# B&R Automation Studio project EFI (part 20)

#### MachineCtrl_Slow.var
```iecst
VAR
	iPrimerBarMechanicalPosition : USINT; (*Position of white bar regarding mechanical assembly*)
	iPrimerBarMapping : USINT; (*Position of white bar regarding printing definition in UI*)
	iWhiteBarMechanicalPosition : USINT; (*Position of white bar regarding mechanical assembly*)
	iWhiteBarMapping : USINT; (*Position of white bar regarding printing definition in UI*)
	arNotLoadedImage : AutoResetSound;
	arSAIFault : AutoResetSound;
	arBentTile : AutoResetSound;
	arPDSensorErrorL1 : AutoResetSound;
	arPDSensorErrorL2 : AutoResetSound;
	xAllBlocksCleaning : BOOL;
	xInstantPrintL2 : BOOL;
	xAllBlocksCleaningEnded : BOOL;
	xInstantPrintL1 : BOOL; (*command bool edge*)
	xShotLine2 : BOOL;
	xCleanSequencially : BOOL := FALSE;
	xShotLine1 : BOOL;
	xOrderToGap : BOOL;
	xCleanBeltForced : BOOL;
	xCleaningBeltByTiles : BOOL;
	xOutputConsentInSingleLineL1 : BOOL;
	xOutputConsentInByPassL1 : BOOL;
	xOutputConsentInByPassL2 : BOOL;
	xOutputConsentInDTPL1 : BOOL;
	xOutputConsentInDTPL2 : BOOL;
	xDoubleLineConsent : BOOL; (*Belt Consent in DobleLine Mode*)
	xOnPcs : BOOL;
	xCleaningBeltByTime : BOOL;
	xCleanBeltOrder : BOOL; (*Internal to assign cleaning belt system *)
	arBlockCleaningEnded : ARRAY[GC_FIRST_BLOCK..MAX_LAST_BLOCK] OF BOOL;
	enCleaningState : CleaningState_enum := CLN_NOT_CLEANING;
	FbCleanDelayControl_1 : FbCleanDelayControl;
	tof_ResetCB1 : TOF;
	xSuctionTurbine : BOOL;
	xEnableCleanBeltMotorMovement : BOOL;
	tp_ToSwapCleanBeltMtrDirection : TP;
	tofCleaningTrayBelt : TOF;
	rsSuction : RS; (*Suction/Mist collector turbine*)
	tofDelaySuction : TOF; (*tiMinutes : TIME;*)
	tof_ResetRouter : TOF;
	tonIntantPrintL2 : TON;
	tonIntantPrintL1 : TON;
	T_ExternalCleaningOrder : TON;
	T_ShotL2Off : TON;
	T_OnPcs : TON;
	ResetCleanBeltCommands : StGeneral_CleanBelt;
	tonCleaningByTime : TON; (*Belt Cleaning*)
	T_ShotL1Off : TON;
	T_OnPC2 : TON;
	T_BtwnCleans : TON;
	tonDelayConsentInput : TON;
	T_OnPC1 : TON;
	tonDelayConsentOutL2 : TON;
	tonDelayConsentOutL1 : TON;
	tonCleaningBelt : TON;
	T_WaitPC2 : TON;
	T_WaitPC1 : TON;
	tonCleanBelt : TON;
	uiSecondsToCleanStop : UDINT; (*Counter of the seconds to clean in the mode*)
	uiSecondsToCleanProd : UDINT; (*Counter of the seconds to clean in the mode*)
	uiSecondsToCleanTotal : UDINT; (*Counter of the seconds to clean in the mode*)
	TP_ShotL1On : TP; (*Careful. It is a TP!!*)
	TP_ShotL2On : TP; (*Careful. It is a TP!!*)
	iIndexCuringLed : USINT;
	iIndexCuringLedLamps : USINT;
	iIndexInks : USINT; (*Inks Index to use a FOR*)
	iIndexBlock : USINT; (*Block Index to use a FOR*)
	xRepetitionLine1 : BOOL;
	xRepetitionLine2 : BOOL;
	iSPTilesToCleanBelt : INT;
	arNoThicknessSystem : AutoResetSound;
	xDelayCleaningOk : BOOL; (*Internal state in printer used on gap and delay line*)
	TNotZero : TON;
	xAnyBlockToPrint : BOOL;
	reasonSoundGen : UDINT;
	reasonSoundGen2 : UDINT;
	reasonSoundInks : UDINT;
	arSAIPowerFault : AutoResetSound;
	arHeaterTankPsu : AutoResetSound;
	xAnyBarLoadedInJob : BOOL; (*Some bar stopped by critical alarm*)
	xAnyInkCriticalAlrm : BOOL; (*Some bar stopped by critical alarm*)
	iIndex : USINT; (*FOR index*)
	iBentTilesCounter : UINT; (*Counter of bent media. Just for the alarm of max movements*)
	tonDecreaseMovCount : TON; (*Time to decrease the count of max movements*)
	tonPCCabinetAlrm : TON;
	tonWasteInkTankMaxLevelReached : TON;
	T_AlarmAir1 : TON;
	xAnyPrintheadsPowered : BOOL;
	xAnyTankHeaterEnabled : BOOL;
	tonStartSound : TON;
	iCountStartSound : USINT;
	xStartSound : BOOL;
	strAux : STRING[80];
	plcCardsOK : ARRAY[0..1] OF UDINT;
	arAlrMountedPiece : AutoResetSound;
	iGroup : USINT;
	stProgramName : STRING[80];
	identInitialize : UDINT;
	iSuspendInit : UINT := 10;
	identAnalogThick : UDINT;
	iResumeAnalogThick : UINT := 10;
	iSuspendAnalogThick : UINT := 10;
	identAnalogFast : UDINT;
	iResumeAnalogFast : UINT := 10;
	iSuspendAnalogFast : UINT := 10;
	identLaserFast : UDINT;
	iResumeLaserFast : UINT := 10;
	iSuspendLaserFast : UINT := 10;
	identLaserCtrl : UDINT;
	iResumeLaserCtrl : UINT := 10;
	iSuspendLaserCtrl : UINT := 10;
	identInitStepper : UDINT;
	iResumeInitStepper : UINT := 10;
	iSuspendInitStepper : UINT := 10;
	identStepper1 : UDINT;
	iResumeStepper1 : UINT := 10;
	iSuspendStepper1 : UINT := 10;
	identStepper2 : UDINT;
	iResumeStepper2 : UINT := 10;
	iSuspendStepper2 : UINT := 10;
	identAxisStepper1 : UDINT;
	iResumeAxisStepper1 : UINT := 10;
	iSuspendAxisStepper1 : UINT := 10;
	identAxisStepper2 : UDINT;
	iResumeAxisStepper2 : UINT := 10;
	iSuspendAxisStepper2 : UINT := 10;
	nResumeAnalog : UDINT;
	nSuspendAnalog : UDINT;
	nResumeLaser : UDINT;
	nSuspendLaser : UDINT;
	nProgramManager : UINT;
	iReasonToSendCleanOrder : USINT;
	tofKeepReliefSignal : TOF;
	iIndexLamps : INT;
	xCleanBeltTopContinue : BOOL;
	xCleanBeltContinue : BOOL;
	xCleanBeltTopForced : BOOL;
	xCleaningBeltTopByTiles : BOOL;
	xCleaningBeltTopByTime : BOOL;
	xCleanBeltTopOrder : BOOL; (*Internal to assign cleaning belt system *)
	tonCleanBeltTopByTime : TON;
	tiCleaningBeltTopByTime : TIME;
	iSPTilesToCleanBeltTop : INT;
	tonCleaningBeltTop : TON;
	tonUpBarsNoConsent : TON;
	tpStoppedMediaInsd : TP;
	BlnkMediaInside : BlinkOnOff;
	arsSwCriticalCondition : AutoResetSound;
	arsWrongDingPos : AutoResetSound;
	statusReset : UINT;
	iPdCalibrationState : INT;
	iPdCalibrationStep : INT;
	iCounter : INT;
	xTeachSignal : BOOL;
	xMarkForTesting : BOOL;
	xBlinkHighPulse : BOOL;
	TON_DelayOutput : TON;
	TON_PDSignal : TON;
	xAvoidRaiseBarsNotConsent : BOOL;
	tonUpsPowerFault : TON;
	iReasonReadyToReset : UINT;
	stEventLogWarningSize : EventLog_typ;
	stEventLogImgLoadedL1 : EventLog_typ;
	stEventLogImgUnLoadedL1 : EventLog_typ;
	stEventLogAlrNotLoadedImage : EventLog_typ;
	stLogAlrImageLoadButNoBarRelated : EventLog_typ;
	ton_MediaValuesIncoherency : TON;
	strAuxEventDesc : STRING[129];
	xCleanBeltMoveFwd : BOOL; (*To move clean brushed to the contrary direction as belt movement*)
	xCleanBeltMoveBwd : BOOL; (*To move clean brushes same direction as belt movement*)
	iIndexHistory : USINT;
	StateHistory : ARRAY[0..iHistoryLines] OF CleaningBeltState_enum;
	iSecondsNoCleaned : UDINT;
END_VAR
VAR CONSTANT
	iHistoryLines : USINT := 20;
END_VAR
VAR
	enCleanBeltUvStep : CleaningBeltState_enum;
	iReasonStopCleanBeltProcess : UINT;
	tiSumTimeToCleanBelt : TIME;
	tiTimeToCleanBelt : TIME;
	tiTimeCounterToCleanBelt : TIME;
	xSwapBrushesMovementDirection : BOOL;
	xReadyToCleanBelt : BOOL;
	xStopBrushes : BOOL;
	iIndexPhysicalConf : USINT;
	cardPlcConfCheck : REFERENCE TO PlcCardMapping;
	iIndexRequirement : USINT;
	xAnyInkBarStarted : BOOL;
	rMaxStartedTempSetPoint : REAL;
	rMaxStartedInkTemp : REAL;
	rMinStartedTempSetPoint : REAL;
	rMinStartedInkTemp : REAL;
	xRunChiller : BOOL;
	iIndexChillersSlow : USINT;
	iIndexInksSlow : USINT;
	arCommsPcPlc : AutoResetSound;
	enStartUpStatus : StartUpStatus_enum := STRUP_NOT_STARTED;
	iIndexStartUp : USINT;
	UnstabInkStartUp : ARRAY[0..MAX_LAST_INK] OF BOOL; (*Inks unstable so long, so automatic startup is cancelled*)
	xInksStoppedWhileStartUp : BOOL;
	xStartUpAnyBarNotStable : BOOL;
	xStartUpAnyBarNotPowered : BOOL;
	xStartUpAnyBarUnstable : BOOL; (*One bar has been unstable for more than 5' and the startup will be cancelled*)
	iIndexBarNotStable : USINT;
	tonStartingInks : TON;
	xPosibleCancel : USINT;
	xRedLight : BOOL;
	xGreenLight : BOOL;
	xYellowLight : BOOL;
	xBlueLight : BOOL;
	xWhiteLight : BOOL;
END_VAR
VAR RETAIN
	DriveUnit : DriveUnitMngr;
END_VAR
VAR
	rBeltDistanceTravelledMmCopy : REAL;
	rBeltDistanceTravelledMm : REAL;
	stEventLogBeltDistanceTravelled : EventLog_typ;
	rBeltPositionMmInitCopy : REAL;
	rBeltPositionMmInit : REAL;
	rBeltPositionMmFinalCopy : REAL;
	rBeltPositionMmFinal : REAL;
	rBeltSpeedInit : REAL;
	xEdge1sec : BOOL;
	tonWaitToCleanRemote : TON;
	iFaultPcPlcAux : INT;
	T_AlarmComPcPlc : TON;
	xColorBarEnabledToPrint : BOOL;
	xWhiteBarEnabledToPrint : BOOL;
	xClearBarEnabledToPrint : BOOL;
	xRunAirCleaner : BOOL;
	tonBlowerNotRunning : TON;
	tonCheckAlarms : TON;
	ResetAlarms : StGeneral_AirCleaner_Alarms;
	tiPrevToCleanWhenPrinterStopped : TIME;
	tiPrevCleaningByTime : TIME;
	iPrevPiecesNumberToCleanL2 : INT;
	iPrevPiecesNumberToCleanL1 : INT;
END_VAR
```

#### Air.st
```iecst
ACTION Air:

	////////////////////////////////////////////////////////////////////////////////////
	// ZERO MODE
	////////////////////////////////////////////////////////////////////////////////////
	TNotZero.IN:=NOT gMachine.St.Mode.xZero;
	TNotZero.PT:=T#500ms;
	TNotZero();
	gMachine.Out.xAirSupply:= TNotZero.Q AND (NOT gMachine.AlSummary.xAlrSafetyCutAir OR gSafetyController.Inputs.xPrinterMaintenanceKey);

END_ACTION
```

#### AirCleaner.st
```iecst
ACTION AirCleaner:

	IF NOT gAirCleaner.Parameters.xInstalled THEN
		gAxisInverter[gAirCleaner.Parameters.iIndex].Orders.PowerOn := FALSE;
		gAxisInverter[gAirCleaner.Parameters.iIndex].Parameters.Velocity := 0;
		gAirCleaner.Alarms := ResetAlarms;
		RETURN;
	ELSE
		gAxisInverter[gAirCleaner.Parameters.iIndex].Orders.PowerOn := NOT gMachine.St.Mode.xZero;
		gAxisInverter[gAirCleaner.Parameters.iIndex].Parameters.Velocity := REAL_TO_UINT(MAX(354.0, (gAirCleaner.ParSw.rDutyCycle * gAirCleaner.Parameters.rMaxSpeed / 100)));

		//Manual
		IF gMachine.St.Mode.xManual THEN
			xRunAirCleaner := gAirCleaner.OrdersSw.xRun;
		//Auto
		ELSIF gMachine.St.Mode.xAuto THEN
			xRunAirCleaner := (gAirCleaner.OrdersSw.xRun) AND (gBelt.states.xRuningBelt);
		ELSE
			xRunAirCleaner := FALSE;
		END_IF

		//Setting commands with the edge of xRun signal
		gAxisInverter[gAirCleaner.Parameters.iIndex].Commands.MovePositive := EDGEPOS(xRunAirCleaner) AND gAirCleaner.Parameters.Direction = MOTOR_POSITIVE;
		gAxisInverter[gAirCleaner.Parameters.iIndex].Commands.MoveNegative := EDGEPOS(xRunAirCleaner) AND gAirCleaner.Parameters.Direction = MOTOR_NEGATIVE;

		//Stop
		gAxisInverter[gAirCleaner.Parameters.iIndex].Commands.Stop := EDGENEG(xRunAirCleaner);

		//Alarms
		IF gAxisInverter[gAirCleaner.Parameters.iIndex].Status.ErrorComms THEN
			gAirCleaner.Alarms.xDriveComms := TRUE;
		END_IF

		tonCheckAlarms.IN := gMachine.In.xSafetyEnabled;
		tonCheckAlarms.PT := T#3000ms;
		tonCheckAlarms();

		//Driver Blower Error
		IF tonCheckAlarms.Q AND NOT gAirCleaner.Alarms.xDriveComms THEN
			IF ((gAxisInverter[gAirCleaner.Parameters.iIndex].Status.ErrorID <> 0) AND (gAxisInverter[gAirCleaner.Parameters.iIndex].Status.ErrorID <> 20625)) OR gAxisInverter[gAirCleaner.Parameters.iIndex].Status.StatusErrorStop THEN
				gAirCleaner.Alarms.xDriveError := TRUE;
			END_IF

			IF NOT gAxisInverter[gAirCleaner.Parameters.iIndex].ElecSignals.In.xBreakerOK THEN
				gAirCleaner.Alarms.xInverterPowerFault := TRUE;
			END_IF
		END_IF

		//Using Orders.PowerOn because Commands.MovePositive and Commands.MoveNegative are just edges
		tonBlowerNotRunning.IN := xRunAirCleaner AND gAxisInverter[gAirCleaner.Parameters.iIndex].Parameters.Velocity > 300.0 AND ABS(gAxisInverter[gAirCleaner.Parameters.iIndex].Status.ActVelocity) < 300.0;
		tonBlowerNotRunning.PT := T#5s;
		tonBlowerNotRunning();
		IF tonBlowerNotRunning.Q THEN
			gAirCleaner.Alarms.xBlowerNotRunning := TRUE;
		END_IF

		//Reset
		IF gMachine.AutoCmd.xReset OR EDGEPOS(gMachine.St.Mode.xZero) THEN
			gAxisInverter[gAirCleaner.Parameters.iIndex].Commands.Reset := TRUE;
			gAirCleaner.Alarms := ResetAlarms;
		END_IF
	END_IF

END_ACTION
```

#### AlarmsSlow.st
```iecst
ACTION AlarmsSlow:

	gMachine.St.Blocks.xAnyBarAndBlockReadyToPrint	:= 	(gBlock[1].parSw.xEnableToPrint AND gBlock[1].Status.iBarsReadyToPrint>0) OR
														(gBlock[2].parSw.xEnableToPrint AND gBlock[2].Status.iBarsReadyToPrint>0);

	// Alarm: Not Bars Enabled. It cannot be removed because is stopping printer if you want print and there is not bar recirculationg
	gMachine.Al.Alarm.xAlarmEnableWithoutBarsOn := 	gMachine.St.Mode.xAuto AND
													NOT gMachine.St.AutoMode.xBypass AND
													NOT gMachine.St.AutoMode.xLaboratory AND
													NOT gMachine.St.Blocks.xAnyBarAndBlockReadyToPrint;

	// Alarm: Platform Incoherence
	gMachine.Al.Alarm.xAlarmPlarformInc:= (gMachine.Pt.MachineModel=NoType) AND NOT gMachine.St.Mode.xZero;

	//Alarm: Thickness detection system no selected or selected more than one
	gMachine.Al.Alarm.xAlrThicknSystemNotSelected := NOT gPhotoCells.status.xInstalled AND NOT gDing.State.xDingInstalled;

	//**********
	//UPS Alarms
	//**********

	// Warning: SAI System Fault
	gMachine.Al.Warning.xSAIFault:= gMachine.In.UPSs[1].xSystemFault OR gMachine.In.UPSs[2].xSystemFault;

	// Warning: SAI ByPass
	gMachine.Al.Warning.xSAIBypass:= 	gMachine.In.UPSs[1].xByPass OR
										gMachine.In.UPSs[2].xByPass OR
										gLine.Inputs.UPSs[1].xByPass OR
										gLine.Inputs.UPSs[2].xByPass;

	// Warning: SAI Low Bat
	gMachine.Al.Warning.xSAILowBat:= 	gMachine.In.UPSs[1].xLowBattery OR
										gMachine.In.UPSs[2].xLowBattery OR
										gLine.Inputs.UPSs[1].xLowBattery OR
										gLine.Inputs.UPSs[2].xLowBattery;

	// Alarm: SAI VAC Fault
	tonUpsPowerFault.IN:=	gMachine.In.UPSs[1].xPowerFault OR
							gMachine.In.UPSs[2].xPowerFault OR
							gLine.Inputs.UPSs[1].xPowerFault OR
							gLine.Inputs.UPSs[2].xPowerFault;

	tonUpsPowerFault.PT:=t#20s;
	tonUpsPowerFault();
	IF tonUpsPowerFault.Q THEN gMachine.Al.Alarm.xAlarmSAIPowerFault := TRUE; END_IF;

	gMachine.Al.Alarm.xNoPowered := NOT gMachine.In.xPowerSwitch;

	//Alarm: Colision Danger, no action
	gMachine.Al.Alarm.xNoActionDangerCollision := gBlock[1].Al.xNoActionDangerCollision OR gBlock[2].Al.xNoActionDangerCollision;

	//Critical Ink alarm summary
	xAnyInkCriticalAlrm:=FALSE;
	//To acknowledge if any ink bar is loaded in job. There have been several cases where "gMachine.St.xRobotReadyToPrint" is active but no ink bar's status "ColorLoadedInJob" is active
	xAnyBarLoadedInJob:=FALSE;
	FOR iIndex:=1 TO MAX_LAST_INK BY 1 DO
		IF gInks[iIndex].AlSummary.xAlarmCritical THEN xAnyInkCriticalAlrm := TRUE; END_IF
		IF gInks[iIndex].status.xColorLoadedInJob THEN xAnyBarLoadedInJob := TRUE; END_IF
	END_FOR

	//////// WARNING xNotLoadedImage
	IF gMachine.parSw.Dtp.xDoubleLine THEN
		IF NOT gThicknessCtrl.status.xNewMediaStackEnabled THEN
			gMachine.St.xRobotReadyToPrint := (gMachine.parSw.Dtp.iModeLine1=GC_DTP_RUN AND gMachine.parSw.Electronics.xRobotReadyL1) OR (gMachine.parSw.Dtp.iModeLine2=GC_DTP_RUN AND gMachine.parSw.Electronics.xRobotReadyL2);
		ELSE
			gMachine.St.xRobotReadyToPrint :=	(gMachine.parSw.Dtp.iModeLine1=GC_DTP_RUN AND gMachine.parSw.Electronics.xRobotReadyL1 AND gThicknessCtrl.status.Stack.iNewMediaLoadedL1 > 0) OR
												(gMachine.parSw.Dtp.iModeLine2=GC_DTP_RUN AND gMachine.parSw.Electronics.xRobotReadyL2 AND gThicknessCtrl.status.Stack.iNewMediaLoadedL2 > 0) ;
		END_IF
	ELSE
		IF NOT gThicknessCtrl.status.xNewMediaStackEnabled THEN
			gMachine.St.xRobotReadyToPrint := gMachine.parSw.Electronics.xRobotReadyL1;
		ELSE
			gMachine.St.xRobotReadyToPrint := gMachine.parSw.Electronics.xRobotReadyL1 AND gThicknessCtrl.status.Stack.iNewMediaLoadedL1 > 0;
		END_IF
	END_IF

	IF EDGEPOS(gMachine.parSw.Electronics.xRobotReadyL1) THEN
		LogImageLoadedL1;
	ELSIF EDGENEG(gMachine.parSw.Electronics.xRobotReadyL1) THEN
		LogImageUnLoadedL1;
	END_IF

	//RAISING THE ALARM
	//[RGP] gMachine.St.xMediaDetected variable replaced by "MediaFiltered" to avoid to active "ImageNotLoaded" alarm when belt is not cleaned
	IF gMachine.St.AutoMode.xProdORLab AND gThicknessCtrl.Outputs.xMediaFiltered AND gBelt.states.xRuningBelt AND NOT gLine.StatusSummary.xEmptyingBelts THEN
		IF NOT gMachine.St.xRobotReadyToPrint THEN
			IF gMachine.Pt.xJobNotReadyIsCritical THEN
				gMachine.Al.Alarm.xNotLoadedImage:= TRUE;
			ELSE
				gMachine.Al.Warning.xNotLoadedImage:= TRUE;
			END_IF

		ELSE
			//Due to issue CUBE-1197
			IF NOT xAnyBarLoadedInJob THEN
				gMachine.Al.Warning.xImageLoadedButNoInkBarRelated:= TRUE;
			END_IF
		END_IF
	END_IF

	//IF State is not RUN, remove alarm
	IF (gMachine.St.AutoMode.xProdORLab AND gMachine.parSw.Dtp.iModeLine1<>GC_DTP_RUN AND gMachine.parSw.Dtp.iModeLine2<>GC_DTP_RUN) THEN
		gMachine.Al.Warning.xNotLoadedImage:= FALSE;
	END_IF

	//IF Robot is OK or not in Production or Laboratory , remove alarm
	IF gMachine.St.xRobotReadyToPrint OR (NOT gMachine.St.AutoMode.xProdORLab AND gMachine.Pt.xControlledByLine) THEN
		gMachine.Al.Warning.xNotLoadedImage:= FALSE;
	END_IF

	IF EDGEPOS(gMachine.Al.Warning.xNotLoadedImage) THEN
		LogAlarmImageNotLoaded;
	END_IF

	IF EDGEPOS(gMachine.Al.Warning.xImageLoadedButNoInkBarRelated) THEN
		LogAlarmImageLoadedButNoInkBarRelated;
	END_IF

	// Warning: Max movemets because bent tile	// Warning: Max movemets because bent tile
	// Warning: Max movemets because bent tile	// Warning: Max movemets because bent tile
	IF EDGEPOS (gMachine.Al.Warning.xBentTile) THEN
		iBentTilesCounter := iBentTilesCounter + 1;
	END_IF

	//If time without any change, decrease the count of movements
	tonDecreaseMovCount.IN := NOT gMachine.Al.Warning.xMaxMovsBentTile AND NOT gMachine.Al.Warning.xBentTile AND NOT tonDecreaseMovCount.Q ;
	tonDecreaseMovCount.PT := T#5m;
	tonDecreaseMovCount();
	IF tonDecreaseMovCount.Q THEN
		//Safety decrease to avoid overflow
		iBentTilesCounter:= UINT_SUB(iBentTilesCounter,1);
	END_IF
	IF EDGEPOS(gMachine.Al.Warning.xMaxMovsBentTile) THEN
		iBentTilesCounter:= 0;
	END_IF

	IF iBentTilesCounter >= gc_diNumMaxManiobrasPDoblada THEN
		gMachine.Al.Warning.xMaxMovsBentTile:=TRUE;
	ELSIF  gMachine.AutoCmd.xReset THEN
		gMachine.Al.Warning.xMaxMovsBentTile:=FALSE;
	END_IF

	// Warning: External Cleaning Activate
	IF gMachine.St.Mode.xAuto AND gMachine.AutoCmd.xCleanningByExtOrder AND NOT gMachine.St.AutoMode.xLaboratory THEN
		gMachine.Al.Warning.xExternalCleanActive:= TRUE;

	ELSIF NOT gMachine.St.Mode.xAuto OR (gMachine.St.Cleaning.enCleaningState = CLN_NOT_CLEANING) THEN
		gMachine.Al.Warning.xExternalCleanActive:= FALSE;
	END_IF

	// PC Cabinet Cooling Sensor Alarm
	tonPCCabinetAlrm.IN:= gMachine.In.xCoolingPCSensorAlrm;
	tonPCCabinetAlrm.PT:= T#30S;
	tonPCCabinetAlrm();
	gMachine.Al.Warning.xPCCabineSensAlrm := tonPCCabinetAlrm.Q;

	// Alarm Air1
	T_AlarmAir1.IN:= NOT gMachine.In.xAirSupply AND gBlockInputs[1].xSiUnitModuleOk;
	T_AlarmAir1.PT:= gc_tiTesperaAlarmaAire;
	T_AlarmAir1();
	gMachine.Al.Alarm.xAlarmAir1:= T_AlarmAir1.Q;

	//Alarm: Heater Tank Power Supply Failure
	IF NOT gMachine.In.xTankHeaterPsuOK AND gMachine.St.Blocks.xAnyTankHeaterEnabled THEN
		gMachine.Al.Alarm.xHeaterTankPsu:= TRUE;
		FOR iIndexInks := 1 TO MAX_LAST_INK BY 1 DO gInks[iIndexInks].Al.xAlrHeaterTankPsu := TRUE; END_FOR
	END_IF

	// Raising alarm of stopped media inside.
	// this is a simple way to reset the alarm. A more proper way to remove the alarm would be to
	// use a distanceVar in Thickness_Pos, but this is quite resource consuming, so this would be delayed
	IF gThicknessCtrl.status.MediaPosition.xMediaInside AND NOT gBelt.states.xRuningBelt AND EDGEPOS(gMachine.AutoCmd.xToSafePosition) THEN
		gMachine.Al.Warning.xMediaStoppedInside := TRUE;
	ELSIF gThicknessCtrl.status.Belt.xBeltEmpty THEN
		gMachine.Al.Warning.xMediaStoppedInside := FALSE;
	END_IF

	// Alarm: xUpNotConsent
	gMachine.Al.Warning.xUpNotConsent:= gMachine.St.Consent.xUpWithNoConsent;

	// Warning: PBF card Not OK
	gMachine.Al.Warning.xPbfCardNotOK := gMachine.St.xWorkingAsPBF AND NOT gMachine.In.xPbfCardOK;

	PsycallConfChecking;

	// Warnings: Uv belt cleaning related
	IF gMachine.Pt.Clean.xCleanBeltForUv THEN
		gMachine.Al.Warning.xCleanBeltRelayFaulted := gMachine.In.CleanBelt.xError;
		gMachine.Al.Warning.xCleanCylinderNotInHighPosition := gMachine.In.CleanBelt.xHighPosition;
		gMachine.Al.Warning.xCleanBeltSystemNotInPosition := gMachine.In.CleanBelt.xOpenGuide;
		gMachine.Al.Warning.xBeltCleanRequired := (tiSumTimeToCleanBelt>=gMachine.parSw.CleanBelt.tiCleaningBeltByTime);
	ELSE
		gMachine.Al.Warning.xCleanBeltRelayFaulted := FALSE;
		gMachine.Al.Warning.xCleanCylinderNotInHighPosition := FALSE;
		gMachine.Al.Warning.xCleanBeltSystemNotInPosition:= FALSE;
		gMachine.Al.Warning.xBeltCleanRequired := FALSE;
	END_IF

	//
	IF NOT gMachine.parSw.Clean.xCleanSystemByPieces AND NOT gMachine.parSw.Clean.xCleanSystemByTime THEN
		gMachine.Al.Warning.xNoCleaningModeEnabled:=TRUE;
	ELSE
		gMachine.Al.Warning.xNoCleaningModeEnabled:=FALSE;
	END_IF

	//Hoopers Powered.Warning
	IF gMachine.In.xHoppersSoftStarterFault AND xSuctionTurbine THEN
		gMachine.Al.Warning.xAlrHoopersSoftStarterFault := TRUE;
	END_IF

	//Overvoltage
	IF gMachine.In.xOvervoltage THEN
		gMachine.Al.Warning.xOvervoltage := TRUE;
	END_IF

	//Antistatic device
	IF gMachine.In.AntiStatic.xIonLevelAlarm AND gMachine.Out.xAntiStaticPOn THEN
		gMachine.Al.Warning.xIonAntiStatic := TRUE;
	END_IF
	IF gMachine.In.AntiStatic.xGenAlarm AND gMachine.Out.xAntiStaticPOn THEN
		gMachine.Al.Warning.xErrorAntiStatic := TRUE;
	END_IF

	tonWasteInkTankMaxLevelReached.IN := gMachine.In.xWasteInkTankMaxLevelReached;
	tonWasteInkTankMaxLevelReached.PT := T#500ms;
	tonWasteInkTankMaxLevelReached();
	IF tonWasteInkTankMaxLevelReached.Q THEN
		gMachine.Al.Warning.xWasteInkTankMaxLevelReached := TRUE;
	END_IF

	// NOZOMITWO-2599 Media limitations not updated when enabling ancillaries
	IF gMachine.parSw.Media.rThickness > gMachine.Pt.Media.rMaxMediaThickness OR gMachine.parSw.Media.rThickness < gMachine.Pt.Media.rMinMediaThickness THEN
		gMachine.Al.Alarm.xAlrThickOutLimits := TRUE;
	END_IF
	IF gMachine.parSw.Media.rLength > gMachine.Pt.Media.iMaxMediaLength OR gMachine.parSw.Media.rLength < gMachine.Pt.Media.iMinMediaLength THEN
		gMachine.Al.Alarm.xAlrLengthOutLimits := TRUE;
	END_IF
	IF gMachine.parSw.Media.rWidth > gMachine.Pt.Media.iMaxMediaWidth OR gMachine.parSw.Media.rWidth < gMachine.Pt.Media.iMinMediaLength THEN
		gMachine.Al.Alarm.xAlrWidthOutLimits := TRUE;
	END_IF

	//Alarms comms with kernel
	AlarmKernelPLCCommsCounter;

END_ACTION

ACTION AlarmKernelPLCCommsCounter:

		// Alarm: Com PC-PLC
	T_AlarmComPcPlc.IN:= gMachine.parSw.iFaultComPcPlc=iFaultPcPlcAux;
	T_AlarmComPcPlc.PT:= T#45S;	//This is changed to 45secs
	T_AlarmComPcPlc();

	IF EDGEPOS (T_AlarmComPcPlc.Q) THEN
		gMachine.Al.Alarm.xAlarmComPcPLC:= TRUE;
	END_IF;

	IF (gMachine.parSw.iFaultComPcPlc<>iFaultPcPlcAux) THEN
		iFaultPcPlcAux:= gMachine.parSw.iFaultComPcPlc;
	END_IF;

END_ACTION

ACTION PsycallConfChecking:
	CASE gMachine.Pt.ConfigNameID OF
		GC_CONFIG_2BK12BAR_ID:
			PhysicalConfCheckingWithCardsArray;

		GC_CONFIG_1BK2BAR_ID:
			CASE gMachine.Pt.MachineModel OF
				Type_SHLD,
				Type_SHLD_L:							// SHIELD 1 Block 2 Bars
					plcCardsOK[0].0 := NOT X20DIF371_001.ModuleOk;
					plcCardsOK[0].1 := NOT X20DIF371_002.ModuleOk;
					plcCardsOK[0].2 := NOT X20DIF371_003.ModuleOk;
					plcCardsOK[0].3 := NOT X20DIF371_004.ModuleOk;
					plcCardsOK[0].4 := NOT X20DOF322_005.ModuleOk;
					plcCardsOK[0].5 := NOT X20DOF322_006.ModuleOk;
					plcCardsOK[0].6 := NOT X20AI4322_008.ModuleOk;
					plcCardsOK[0].7 := NOT X20AO4622_009.ModuleOk;
					plcCardsOK[0].8 := NOT X20AT4222_010.ModuleOk;
					plcCardsOK[0].9 :=	NOT gPhotoCells.status.xBackModuleOk;
					plcCardsOK[0].10 := NOT gPhotoCells.status.xFrontModuleOk;

						gMachine.Al.Alarm.xAlrWrongPhysConf := plcCardsOK[0]<>0;

				ELSE
					gMachine.Al.Alarm.xAlrWrongPhysConf := TRUE;

			END_CASE

		GC_CONFIG_BM_1BK8BAR_ID:
			CASE gMachine.Pt.MachineModel OF
				Type_S1400,
				Type_P5_OIL,
				Type_P5_WTR:										//S1400 Without vacuunm
					plcCardsOK[0].0 := NOT X20DIF371_001.ModuleOk;
					plcCardsOK[0].1 := NOT X20DIF371_002.ModuleOk;
					plcCardsOK[0].2 := NOT X20DIF371_003.ModuleOk;
					plcCardsOK[0].3 := NOT X20DIF371_004.ModuleOk;
					plcCardsOK[0].4 := NOT X20DIF371_005.ModuleOk;
					plcCardsOK[0].5 := NOT X20DIF371_006.ModuleOk;
					plcCardsOK[0].6 := NOT X20DI9372_008.ModuleOk;
					plcCardsOK[0].7 := NOT X20DOF322_009.ModuleOk;
					plcCardsOK[0].8 := NOT X20DOF322_010.ModuleOk;
					plcCardsOK[0].9 := NOT X20DOF322_011.ModuleOk;
					plcCardsOK[0].10 := NOT X20DOF322_012.ModuleOk;
					plcCardsOK[0].11 := NOT X20DOF322_013.ModuleOk;
					plcCardsOK[0].12 := NOT X20AI8321_015.ModuleOk;
					plcCardsOK[0].13 := NOT X20AI8321_016.ModuleOk;
					plcCardsOK[0].14 := NOT X20AO4622_017.ModuleOk;
					plcCardsOK[0].15 := NOT X20AO4622_018.ModuleOk;
					plcCardsOK[0].16 := NOT X20AO4622_019.ModuleOk;
					plcCardsOK[0].17:= NOT X20AO4622_020.ModuleOk;
					plcCardsOK[0].18 := NOT X20AT4222_022.ModuleOk;
					plcCardsOK[0].19 := NOT X20AT4222_023.ModuleOk;

				Type_S1400_VAC_PWRLNK,
				Type_S1400_VAC_CAN:							//S1400 With Vacuum
					plcCardsOK[0].0 := NOT X20DIF371_001.ModuleOk;
					plcCardsOK[0].1 := NOT X20DIF371_002.ModuleOk;
					plcCardsOK[0].2 := NOT X20DIF371_003.ModuleOk;
					plcCardsOK[0].3 := NOT X20DIF371_004.ModuleOk;
					plcCardsOK[0].4 := NOT X20DIF371_005.ModuleOk;
					plcCardsOK[0].5 := NOT X20DIF371_006.ModuleOk;
					plcCardsOK[0].6 := NOT X20DI9372_008.ModuleOk;
					plcCardsOK[0].7 := NOT X20DOF322_009.ModuleOk;
					plcCardsOK[0].8 := NOT X20DOF322_010.ModuleOk;
					plcCardsOK[0].9 := NOT X20DOF322_011.ModuleOk;
					plcCardsOK[0].10 := NOT X20DOF322_012.ModuleOk;
					plcCardsOK[0].11 := NOT X20DOF322_013.ModuleOk;
					plcCardsOK[0].12 := NOT X20AI8321_015.ModuleOk;
					plcCardsOK[0].13 := NOT X20AI8321_016.ModuleOk;
					plcCardsOK[0].14 := NOT X20AO4622_017.ModuleOk;
					plcCardsOK[0].15 := NOT X20AO4622_018.ModuleOk;
					plcCardsOK[0].16 := NOT X20AO4622_019.ModuleOk;
					plcCardsOK[0].17 := NOT X20AO4622_020.ModuleOk;
					plcCardsOK[0].18 := NOT X20AT4222_022.ModuleOk;
					plcCardsOK[0].19 := NOT X20AT4222_023.ModuleOk;
					plcCardsOK[0].20 := NOT X20DIF371_024.ModuleOk;
					plcCardsOK[0].21 := NOT X20AI8321_025.ModuleOk;
					plcCardsOK[0].22 := NOT X20AI2636_100.ModuleOk;

					gMachine.Al.Alarm.xAlrWrongPhysConf := plcCardsOK[0]<>0;
				ELSE
					gMachine.Al.Alarm.xAlrWrongPhysConf := TRUE;
			END_CASE

		GC_CONFIG_1BK8BAR_NOZ2_ID,
		GC_CONFIG_1BK8BAR_NOZ2_AQ_ID:
			CASE gMachine.Pt.MachineModel OF
				Type_NOZ_2_AQ:

					//Printer
					plcCardsOK[0].0 := NOT X20DIF371_101.ModuleOk;
					plcCardsOK[0].1 := NOT X20DIF371_102.ModuleOk;
					plcCardsOK[0].2 := NOT X20DIF371_103.ModuleOk;
					plcCardsOK[0].3 := NOT X20DIF371_104.ModuleOk;
					plcCardsOK[0].4 := NOT X20DIF371_105.ModuleOk;
					//plcCardsOK[0].5 := NOT X20PS3300_106.ModuleOk;
					plcCardsOK[0].6 := NOT X20DI9372_107.ModuleOk;
					plcCardsOK[0].7 := NOT X20DOF322_108.ModuleOk;
					plcCardsOK[0].8 := NOT X20DOF322_109.ModuleOk;
					plcCardsOK[0].9 := NOT X20DOF322_110.ModuleOk;
					plcCardsOK[0].10 := NOT X20AI8321_111.ModuleOk;
					plcCardsOK[0].11 := NOT X20AI8321_112.ModuleOk;
					plcCardsOK[0].12 := NOT X20AI8321_113.ModuleOk;
					//plcCardsOK[0].13 := NOT X20PS3300_114.ModuleOk;
					plcCardsOK[0].14 := NOT X20AO4622_115.ModuleOk;
					plcCardsOK[0].15 := NOT X20AO4622_116.ModuleOk;
					plcCardsOK[0].16 := NOT X20AO4622_117.ModuleOk;
					plcCardsOK[0].17:= NOT X20AT4222_118.ModuleOk;
					plcCardsOK[0].18 := NOT X20AT4222_119.ModuleOk;

					//PDC
					plcCardsOK[1].0 := NOT Pdc_X20DIF371_002.ModuleOk;
					plcCardsOK[1].1 := NOT Pdc_X20DIF371_003.ModuleOk;
					plcCardsOK[1].2 := NOT Pdc_X20DIF371_004.ModuleOk;
					plcCardsOK[1].3 := NOT Pdc_X20DIF371_005.ModuleOk;
					plcCardsOK[1].4 := NOT Pdc_X20DIF371_006.ModuleOk;
					plcCardsOK[1].5 := NOT X20PS3300_007.ModuleOk;
					plcCardsOK[1].6 := NOT Pdc_X20DOF322_008.ModuleOk;
					plcCardsOK[1].7 := NOT Pdc_X20DOF322_009.ModuleOk;
					plcCardsOK[1].8 := NOT Pdc_X20DOF322_010.ModuleOk;

					gMachine.Al.Alarm.xAlrWrongPhysConf := plcCardsOK[0]<>0 OR plcCardsOK[1]<>0;

				Type_NOZ_2_UV,
				Type_NOZ_2_UV_White:

					//Printer
					plcCardsOK[0].0 := NOT X20DIF371_101.ModuleOk;
					plcCardsOK[0].1 := NOT X20DIF371_102.ModuleOk;
					plcCardsOK[0].2 := NOT X20DIF371_103.ModuleOk;
					plcCardsOK[0].3 := NOT X20DIF371_104.ModuleOk;
					plcCardsOK[0].4 := NOT X20DIF371_105.ModuleOk;
					plcCardsOK[0].5 := NOT X20PS3300_106.ModuleOk;
					plcCardsOK[0].6 := NOT X20DI9372_107.ModuleOk;
					plcCardsOK[0].7 := NOT X20DOF322_108.ModuleOk;
					plcCardsOK[0].8 := NOT X20DOF322_109.ModuleOk;
					plcCardsOK[0].9 := NOT X20DOF322_110.ModuleOk;
					plcCardsOK[0].10 := NOT X20AI8321_111.ModuleOk;
					plcCardsOK[0].11 := NOT X20AI8321_112.ModuleOk;
					plcCardsOK[0].12 := NOT X20AI8321_113.ModuleOk;
					plcCardsOK[0].13 := NOT X20PS3300_114.ModuleOk;
					plcCardsOK[0].14 := NOT X20AO4622_115.ModuleOk;
					plcCardsOK[0].15 := NOT X20AO4622_116.ModuleOk;
					plcCardsOK[0].16 := NOT X20AO4622_117.ModuleOk;
					plcCardsOK[0].17:= NOT X20AT4222_118.ModuleOk;
					plcCardsOK[0].18 := NOT X20AT4222_119.ModuleOk;
					//plcCardsOK[0].19 := NOT X20CS1030_150.ModuleOk;
					//plcCardsOK[0].20 := NOT X20CS1030_151.ModuleOk;
					plcCardsOK[0].21 := NOT X20PS3300_152.ModuleOk;
					plcCardsOK[0].22 := NOT X20DIF371_153.ModuleOk;
					plcCardsOK[0].23 := NOT X20DIF371_154.ModuleOk;
					plcCardsOK[0].24 := NOT X20DOF322_155.ModuleOk;
					plcCardsOK[0].25 := NOT X20AI8221_156.ModuleOk;
					plcCardsOK[0].26 := NOT X20AO4622_157.ModuleOk;
					plcCardsOK[0].27 := NOT X20AO4622_158.ModuleOk;

					//PDC
					plcCardsOK[1].0 := NOT Pdc_X20DIF371_002.ModuleOk;
					plcCardsOK[1].1 := NOT Pdc_X20DIF371_003.ModuleOk;
					plcCardsOK[1].2 := NOT Pdc_X20DIF371_004.ModuleOk;
					plcCardsOK[1].3 := NOT Pdc_X20DIF371_005.ModuleOk;
					plcCardsOK[1].4 := NOT Pdc_X20DIF371_006.ModuleOk;
					plcCardsOK[1].5 := NOT X20PS3300_007.ModuleOk;
					plcCardsOK[1].6 := NOT Pdc_X20DOF322_008.ModuleOk;
					plcCardsOK[1].7 := NOT Pdc_X20DOF322_009.ModuleOk;
					plcCardsOK[1].8 := NOT Pdc_X20DOF322_010.ModuleOk;
					plcCardsOK[1].9 := NOT Pdc_X20DIF371_020.ModuleOk;
					plcCardsOK[1].10 := NOT Pdc_X20DIF371_021.ModuleOk;
					plcCardsOK[1].11 := NOT X20PS3300_022.ModuleOk;
					plcCardsOK[1].12 := NOT Pdc_X20DOF322_023.ModuleOk;

					gMachine.Al.Alarm.xAlrWrongPhysConf := plcCardsOK[0]<>0 OR plcCardsOK[1]<>0;

				ELSE
					gMachine.Al.Alarm.xAlrWrongPhysConf := TRUE;

			END_CASE

		GC_CONFIG_1BK7BAR_CUBE_ID:
			plcCardsOK[0].0 := NOT X20DIF371_101.ModuleOk;
			plcCardsOK[0].1 := NOT X20DIF371_102.ModuleOk;
			plcCardsOK[0].2 := NOT X20DIF371_103.ModuleOk;
			plcCardsOK[0].3 := NOT X20DIF371_104.ModuleOk;
			plcCardsOK[0].4 := NOT X20PS3300_106.ModuleOk;
			plcCardsOK[0].5 := NOT X20DOF322_108.ModuleOk;
			plcCardsOK[0].6 := NOT X20DOF322_109.ModuleOk;
			plcCardsOK[0].7 := NOT X20AI8321_111.ModuleOk;
			plcCardsOK[0].8 := NOT X20AI8321_112.ModuleOk;
			plcCardsOK[0].9 := NOT X20AI8321_113.ModuleOk;
			plcCardsOK[0].10 := NOT X20PS3300_114.ModuleOk;
			plcCardsOK[0].11 := NOT X20AO4622_115.ModuleOk;
			plcCardsOK[0].12 := NOT X20AO4622_116.ModuleOk;
			plcCardsOK[0].13 := NOT X20AO4622_117.ModuleOk;
			plcCardsOK[0].14 := NOT X20AO4622_118.ModuleOk;
			plcCardsOK[0].15 := NOT X20AT4222_119.ModuleOk;
			plcCardsOK[0].16 := NOT X20AT4222_120.ModuleOk;
			plcCardsOK[0].17 := NOT X20CS1030_121.ModuleOk;
			//plcCardsOK[0].18 := NOT X20DI9372_140.ModuleOk;

			//PDC
			plcCardsOK[1].1 := NOT Pdc_X20DIF371_002.ModuleOk;
			plcCardsOK[1].2 := NOT Pdc_X20DIF371_003.ModuleOk;
			plcCardsOK[1].3 := NOT Pdc_X20DIF371_004.ModuleOk;
			plcCardsOK[1].4 := NOT Pdc_X20DOF322_005.ModuleOk;
			plcCardsOK[1].5 := NOT X20PS3300_006.ModuleOk;
			plcCardsOK[1].6 := NOT Pdc_X20DOF322_007.ModuleOk;
			plcCardsOK[1].7 := NOT Pdc_X20DOF322_008.ModuleOk;
			plcCardsOK[1].8 := NOT Pdc_X20DIF371_030.ModuleOk;
			plcCardsOK[1].9 := NOT Pdc_X20AI2636_050.ModuleOk;

			gMachine.Al.Alarm.xAlrWrongPhysConf := plcCardsOK[0]<>0 OR plcCardsOK[1]<>0;

		GC_CONFIG_1BK10BAR_MECANO_ID:
			plcCardsOK[0].0 := NOT X20DIF371_101.ModuleOk;
			plcCardsOK[0].1 := NOT X20DIF371_102.ModuleOk;
			plcCardsOK[0].2 := NOT X20DIF371_103.ModuleOk;
			plcCardsOK[0].3 := NOT X20DIF371_104.ModuleOk;
			plcCardsOK[0].4 := NOT X20DIF371_105.ModuleOk;
			plcCardsOK[0].5 := NOT X20DIF371_106.ModuleOk;
			plcCardsOK[0].6 := NOT X20PS3300_107.ModuleOk;
			plcCardsOK[0].7 := NOT X20DOF322_108.ModuleOk;
			plcCardsOK[0].8 := NOT X20DOF322_109.ModuleOk;
			plcCardsOK[0].9 := NOT X20DOF322_110.ModuleOk;
			plcCardsOK[0].10 := NOT X20AI8321_111.ModuleOk;
			plcCardsOK[0].11 := NOT X20AI8321_112.ModuleOk;
			plcCardsOK[0].12 := NOT X20AI8321_113.ModuleOk;
			plcCardsOK[0].13 := NOT X20AI8321_114.ModuleOk;
			plcCardsOK[0].14 := NOT X20PS3300_115.ModuleOk;
			plcCardsOK[0].15 := NOT X20AO4622_116.ModuleOk;
			plcCardsOK[0].16 := NOT X20AO4622_117.ModuleOk;
			plcCardsOK[0].17 := NOT X20AO4622_118.ModuleOk;
			plcCardsOK[0].18 := NOT X20AO4622_119.ModuleOk;
			plcCardsOK[0].19:= NOT X20AT4222_120.ModuleOk;
			plcCardsOK[0].20 := NOT X20AT4222_121.ModuleOk;
			plcCardsOK[0].21 := NOT X20PS3300_150.ModuleOk;
			plcCardsOK[0].22 := NOT X20DIF371_151.ModuleOk;
			plcCardsOK[0].23 := NOT X20DIF371_152.ModuleOk;
			plcCardsOK[0].24 := NOT X20DIF371_153.ModuleOk;
			plcCardsOK[0].25 := NOT X20DIF371_154.ModuleOk;
			plcCardsOK[0].26 := NOT X20DOF322_155.ModuleOk;
			plcCardsOK[0].27 := NOT X20DOF322_156.ModuleOk;
			plcCardsOK[0].28 := NOT X20PS3300_157.ModuleOk;
			plcCardsOK[0].29 := NOT X20AO4622_158.ModuleOk;
			plcCardsOK[0].30 := NOT X20AO4622_159.ModuleOk;
			plcCardsOK[0].31 := NOT X20AO4622_160.ModuleOk;
			plcCardsOK[1].0 := NOT X20AO4622_161.ModuleOk;
			plcCardsOK[1].1 := NOT X20CS1030_162.ModuleOk;
//			IF gMachine.Pt.MachineModel<>Type_MECANO_UV_OPV THEN
//				plcCardsOK[1].2 := NOT X20CS1030_180.ModuleOk;
//			END_IF
//			IF gMachine.Pt.MachineModel<>Type_MECANO_UV_WHITE THEN
//				plcCardsOK[1].3 := NOT X20CS1030_181.ModuleOk;
//			END_IF

			//PDC
			plcCardsOK[1].4 := NOT Pdc_X20DIF371_002.ModuleOk;
			plcCardsOK[1].5 := NOT Pdc_X20DIF371_003.ModuleOk;
			plcCardsOK[1].6 := NOT Pdc_X20DIF371_004.ModuleOk;
			plcCardsOK[1].7 := NOT Pdc_X20DIF371_005.ModuleOk;
			plcCardsOK[1].8 := NOT Pdc_X20DIF371_006.ModuleOk;
			plcCardsOK[1].9 := NOT Pdc_X20DIF371_007.ModuleOk;
			plcCardsOK[1].10 := NOT X20PS3300_008.ModuleOk;
			plcCardsOK[1].11 := NOT Pdc_X20DOF322_009.ModuleOk;
			plcCardsOK[1].12 := NOT Pdc_X20DOF322_010.ModuleOk;
			plcCardsOK[1].13 := NOT Pdc_X20DOF322_011.ModuleOk;
			plcCardsOK[1].14 := NOT X20PS3300_020.ModuleOk;
			plcCardsOK[1].15 := NOT Pdc_X20DIF371_021.ModuleOk;
			plcCardsOK[1].16 := NOT Pdc_X20DIF371_022.ModuleOk;
			plcCardsOK[1].17 := NOT Pdc_X20DIF371_023.ModuleOk;
			plcCardsOK[1].18 := NOT Pdc_X20DIF371_024.ModuleOk;
			plcCardsOK[1].19 := NOT Pdc_X20DOF322_025.ModuleOk;

			gMachine.Al.Alarm.xAlrWrongPhysConf := plcCardsOK[0]<>0 OR plcCardsOK[1]<>0;

		GC_CONFIG_SIMTEST_ID:
			gMachine.Al.Alarm.xAlrWrongPhysConf := FALSE;

		ELSE

			gMachine.Al.Alarm.xAlrWrongPhysConf := TRUE;

	END_CASE

END_ACTION

ACTION PhysicalConfCheckingWithCardsArray:

	// If not assigned, just skip the code
	IF gPlcCards[iIndexPhysicalConf].pCard = 0 THEN
		RETURN;
	END_IF

	cardPlcConfCheck ACCESS gPlcCards[iIndexPhysicalConf].pCard;

	// If the cards is not OK, ckeck if it is needed
	IF NOT cardPlcConfCheck.ModuleOk THEN
		RaisePhysicalConfAlarmIfRequired;
	END_IF

	// Go to next card
	iIndexPhysicalConf := iIndexPhysicalConf + 1;
	IF gPlcCards[iIndexPhysicalConf].Type = CARD_UNDEFINED THEN
		iIndexPhysicalConf := 0;
	END_IF

END_ACTION

ACTION RaisePhysicalConfAlarmIfRequired:

	FOR iIndexRequirement := 0 TO MAX_LAST_REQUIRED_FUNCTION_CARD DO
		CASE gPlcCards[iIndexPhysicalConf].RequiredForFunctions[iIndexRequirement] OF
			CARDREQUIRED_UNDEFINED:
				//Do nothing

			CARDREQUIRED_ALWAYS:
				gMachine.Al.Alarm.xAlrWrongPhysConf := TRUE;

			CARDREQUIRED_ANALOG_THICK:
				IF gDing.State.xDingInstalled THEN
					gMachine.Al.Alarm.xAlrWrongPhysConf := TRUE;
				END_IF

			CARDREQUIRED_SENSOR_THICK:
				IF gPhotoCells.status.xInstalled THEN
					gMachine.Al.Alarm.xAlrWrongPhysConf := TRUE;
				END_IF

			CARDREQUIRED_VACUUM:
				IF gTransVacuum[1].Status.xInstalled THEN
					gMachine.Al.Alarm.xAlrWrongPhysConf := TRUE;
				END_IF

			CARDREQUIRED_LED_WHITE:
				IF gCuringLed[iIndexWhiteCuringLedBar].Status.xInstalled THEN
					gMachine.Al.Alarm.xAlrWrongPhysConf := TRUE;
				END_IF

			CARDREQUIRED_LED_COLOR:
				IF gCuringLed[iIndexColorCuringLedBar].Status.xInstalled THEN
					gMachine.Al.Alarm.xAlrWrongPhysConf := TRUE;
				END_IF

			CARDREQUIRED_HEATED_TANKS:
				IF gMachine.St.Blocks.xAnyTankHeaterEnabled THEN
					gMachine.Al.Alarm.xAlrWrongPhysConf := TRUE;
				END_IF

		END_CASE

	END_FOR

END_ACTION
```

#### BeltShot.st
```iecst
ACTION BeltShot:

	///////////////////////////////////////////////////////////////////////////////////////////////////////////////////////////////////////////////
	///////////////////////////////////////////////// ENABLE SHOTS FROM PLC  //////////////////////////////////////////////////////////////////////
	///////////////////////////////////////////////////////////////////////////////////////////////////////////////////////////////////////////////
	// TOJC: It has to be moved out of here	because commands cannot be updated as commands at the same program.
	// All commands are coming from upper subsystem
	////////////////////////////////////////////////////////////////////////////////////////////////////////////
	// conditions to have enabled shots from PLC set a status
	//
	// Check commandBool Commands received from SW:
	// gui_i_iCmdDisparoL1 OR gui_i_iCmdDisparoL2
	// gui_i_iCmdRepeticionDisparoL1 and gui_i_iCmdRepeticionDisparoL2

	///////////////////////////////////////////////////////////////////////////////////////////////////////////////////////////////////////////////
	///////////////////////////////////////////////// INSTANT AND CONTINUOUS PRINT L1 /////////////////////////////////////////////////////////////
	///////////////////////////////////////////////////////////////////////////////////////////////////////////////////////////////////////////////

	IF gMachine.parSw.Shot.xShotLine1 AND NOT gMachine.parSw.Shot.xRepetitionShotLine1 THEN
		xInstantPrintL1:=TRUE;
	ELSIF tonIntantPrintL1.Q OR gMachine.parSw.Shot.xRepetitionShotLine1 THEN
		xInstantPrintL1:=FALSE;
	END_IF
	tonIntantPrintL1.IN:=xInstantPrintL1;
	tonIntantPrintL1.PT:= T#200MS;
	tonIntantPrintL1();

	///////////////////////////////////////////////////////////////////////////////////////////////////////////////////////////////////////////////
	///////////////////////////////////////////////// SHOTING PRINT L1 ////////////////////////////////////////////////////////////////////////////
	///////////////////////////////////////////////////////////////////////////////////////////////////////////////////////////////////////////////

	// Shooting Line 1
	xRepetitionLine1:= gMachine.parSw.Shot.xRepetitionShotLine1 AND gMachine.St.Position.xInPrint;
	TP_ShotL1On.IN:= xRepetitionLine1 AND NOT T_ShotL1Off.Q;
	TP_ShotL1On.PT:= T#200ms;
	TP_ShotL1On();

	T_ShotL1Off.IN:= gMachine.parSw.Shot.xRepetitionShotLine1 AND NOT T_ShotL1Off.Q;
	T_ShotL1Off.PT:= MAX(gMachine.parSw.Shot.tiShotL1, SHOT_MIN_TIME_BETWEEN_SHOTS);
	T_ShotL1Off();

	//Activation of the output due to an instant print or a continuous print
	xShotLine1	:= xInstantPrintL1 OR TP_ShotL1On.Q;

	//Activation of the outputs
	gBlock[1].Out.xShotLine1 := xShotLine1;
	gBlock[2].Out.xShotLine1 := xShotLine1;

	gMachine.Out.xShotLine1 := xShotLine1;

	///////////////////////////////////////////////////////////////////////////////////////////////////////////////////////////////////////////////
	///////////////////////////////////////////////// INSTANT AND CONTINUOUS PRINT L2 /////////////////////////////////////////////////////////////
	///////////////////////////////////////////////////////////////////////////////////////////////////////////////////////////////////////////////

	IF gMachine.parSw.Shot.xShotLine2 AND NOT gMachine.parSw.Shot.xRepetitionShotLine2 THEN
		xInstantPrintL2:=TRUE;
	ELSIF tonIntantPrintL2.Q OR gMachine.parSw.Shot.xRepetitionShotLine2 THEN
		xInstantPrintL2:=FALSE;
	END_IF
	tonIntantPrintL2.IN:=xInstantPrintL2;
	tonIntantPrintL2.PT:= T#200MS;
	tonIntantPrintL2();

	///////////////////////////////////////////////////////////////////////////////////////////////////////////////////////////////////////////////
	///////////////////////////////////////////////// SHOTING PRINT L2 ////////////////////////////////////////////////////////////////////////////
	///////////////////////////////////////////////////////////////////////////////////////////////////////////////////////////////////////////////

	// Shooting Line 2
	xRepetitionLine2:= gMachine.parSw.Shot.xRepetitionShotLine2 AND gMachine.St.Position.xInPrint;
	TP_ShotL2On.IN:= xRepetitionLine2 AND NOT T_ShotL2Off.Q;
	TP_ShotL2On.PT:= T#200ms;
	TP_ShotL2On();

	T_ShotL2Off.IN:= gMachine.parSw.Shot.xRepetitionShotLine2 AND NOT T_ShotL2Off.Q;
	T_ShotL2Off.PT:= MAX(gMachine.parSw.Shot.tiShotL2, SHOT_MIN_TIME_BETWEEN_SHOTS);
	T_ShotL2Off();

	//Activation of the output due to an instant print or a continuous print
	xShotLine2	:= xInstantPrintL2 OR TP_ShotL2On.Q;

	//Activation of the outputs
	gBlock[1].Out.xShotLine2 := xShotLine2;
	gBlock[2].Out.xShotLine2 := xShotLine2;

	gMachine.Out.xShotLine2 := xShotLine2;

	//Remove Edge commands to Use them just as Edge
	gMachine.parSw.Shot.xShotLine1 := FALSE;
	gMachine.parSw.Shot.xShotLine2 := FALSE;

END_ACTION
```

#### CheckValues.st
```iecst
ACTION CheckValues:

	// MEDIA // MEDIA // MEDIA // MEDIA // MEDIA // MEDIA // MEDIA
	// MEDIA // MEDIA // MEDIA // MEDIA // MEDIA // MEDIA // MEDIA

	IF NOT gMachine.parSw.Dtp.xDoubleLine THEN
		// Single line check
		CheckSingleLineMedia;
	END_IF

END_ACTION

ACTION CheckSingleLineMedia:

	//The Maximum width is 1400, So 2*Offset + Width should always be 1400. If no, it is an error of the values from Sw
	ton_MediaValuesIncoherency.IN := 2 * gMachine.parSw.Media.rOffsetRegisterL1 + gMachine.parSw.Media.rWidth < 1395;
	ton_MediaValuesIncoherency.PT := T#200ms;
	ton_MediaValuesIncoherency();

	// If the values are consistent in time, raise and log the message
	IF EDGEPOS(ton_MediaValuesIncoherency.Q) THEN
		LogWarningSize;

		// Avoid non curing media by setting the maximum width
		//gMachine.parSw.Media.rOffsetRegisterL1 := 1;
		//gMachine.parSw.Media.rWidth := 1400;
	END_IF

END_ACTION
```

#### CleanBeltUv.st
```iecst
ACTION CleanBeltUv:

	///////////////////////////////////////////////////////////////////////////////////////////////////////////////////
	// General conditions to clean belt	when machine is in AUTOMATIC OR MANUAL MODES
	///////////////////////////////////////////////////////////////////////////////////////////////////////////////////

	//Delay falling the tray to be sure no water is poured inside the machine
	tofCleaningTrayBelt.IN:=gBelt.states.xRuningBelt;
	tofCleaningTrayBelt.PT:=T#200MS;
	tofCleaningTrayBelt();

	IF gBelt.states.xRuningBelt AND gMachine.parSw.CleanBelt.xCleanBeltByTime AND gMachine.St.Position.xInPrint THEN
		IF EDGEPOS(gPLC.xBlk_500ms) THEN
			tiSumTimeToCleanBelt:=tiSumTimeToCleanBelt + INT_TO_TIME(1000); //Time in seconds
		END_IF
	END_IF

	xCleanBeltOrder := gMachine.AutoCmd.xCleanBelt;
	xSwapBrushesMovementDirection := gThicknessCtrl.status.Belt.iBeltTurns>=gMachine.parSw.CleanBelt.iBeltTurns;
	xStopBrushes := (2*gMachine.parSw.CleanBelt.iBeltTurns)=gThicknessCtrl.status.Belt.iBeltTurns;

	xReadyToCleanBelt := NOT gBelt.states.xRuningBelt AND ((gMachine.St.AutoMode.xStop AND NOT gMachine.Pt.xControlledByLine) OR
															gLine.StatusSummary.xIdle);

	//Cleaning process states
	CASE enCleanBeltUvStep OF

		//Out of automatic mode
		CLN_BELT_NOT_READY:
			gMachine.commands.xRunBelt := FALSE;
			xCleanBeltMoveFwd := FALSE;
			xCleanBeltMoveBwd := FALSE;
			IF xReadyToCleanBelt AND NOT gMachine.In.CleanBelt.xOpenGuide THEN
				enCleanBeltUvStep := CLN_BELT_READY_TO_CLEAN;
			END_IF

		//Machine in auto and stopped
		CLN_BELT_READY_TO_CLEAN:
			IF xCleanBeltOrder THEN
				enCleanBeltUvStep := CLN_BELT_CLEANING_START;
			END_IF

		//Run belt
		CLN_BELT_CLEANING_START:
			gMachine.commands.xRunBelt := TRUE;
			IF gBelt.states.xRuningBelt THEN
				enCleanBeltUvStep := CLN_BELT_CLEAN_CLOKWISE;
			END_IF

		//Run brushes clockwise
		CLN_BELT_CLEAN_CLOKWISE:
			xCleanBeltMoveFwd := TRUE;
			IF xSwapBrushesMovementDirection THEN
				xCleanBeltMoveFwd := FALSE;
				enCleanBeltUvStep := CLN_BELT_CLEAN_COUNTERCLOCKWISE;
			END_IF

		//Run brushes counterclockwise
		CLN_BELT_CLEAN_COUNTERCLOCKWISE:
			xCleanBeltMoveBwd := TRUE;
			IF xStopBrushes THEN
				xCleanBeltMoveBwd := FALSE;
				enCleanBeltUvStep := CLN_BELT_CLEANED;
			END_IF

		//Stop belt
		CLN_BELT_CLEANED:
			tiSumTimeToCleanBelt:=0;
			gMachine.commands.xRunBelt := FALSE;
			IF NOT gBelt.states.xRuningBelt THEN
				enCleanBeltUvStep := CLN_BELT_NOT_READY;
			END_IF

		//Process error
		CLN_BELT_ERROR:
			gMachine.commands.xRunBelt := FALSE;
			xCleanBeltMoveFwd := FALSE;
			xCleanBeltMoveBwd := FALSE;
			IF iReasonStopCleanBeltProcess=0 THEN
				enCleanBeltUvStep := CLN_BELT_NOT_READY;
			END_IF
	END_CASE

	//To
	iReasonStopCleanBeltProcess.0 := gMachine.AlSummary.xAlarmStop;
	iReasonStopCleanBeltProcess.1 := gMachine.AlSummary.xAlarmCritical;
	iReasonStopCleanBeltProcess.2 := NOT gMachine.St.Mode.xAuto;
	iReasonStopCleanBeltProcess.3 := gMachine.In.Buttons.xStop;
	IF iReasonStopCleanBeltProcess>0 THEN
		enCleanBeltUvStep := CLN_BELT_ERROR;

//	ELSIF NOT xReadyToCleanBelt THEN
//		enCleanBeltUvStep := CLN_BELT_NOT_READY;
	END_IF

	//Store the history of the status to easy the debug
	IF enCleanBeltUvStep<>StateHistory[0] THEN
		FOR iIndexHistory:=iHistoryLines TO 1 BY -1 DO
			StateHistory[iIndexHistory]:=StateHistory[iIndexHistory-1];
		END_FOR;
		StateHistory[0]:=enCleanBeltUvStep;
	END_IF

	tiTimeToCleanBelt:= LIMIT(0, (gMachine.parSw.CleanBelt.tiCleaningBeltByTime-tiSumTimeToCleanBelt), gMachine.parSw.CleanBelt.tiCleaningBeltByTime); //Time in ms
	gMachine.St.CleaningBelt.iTimeToCleanBelt := TIME_TO_INT(tiTimeToCleanBelt/(60*1000)); //Time in minutes
	gMachine.St.CleaningBelt.enState := enCleanBeltUvStep;
	gMachine.St.CleaningBelt.xCleaningProcessOnGoing := enCleanBeltUvStep=CLN_BELT_CLEANING_START OR
														enCleanBeltUvStep=CLN_BELT_CLEAN_CLOKWISE OR
														enCleanBeltUvStep=CLN_BELT_CLEAN_COUNTERCLOCKWISE OR
														enCleanBeltUvStep=CLN_BELT_CLEANED;

	//This variable will be read by Sw to show a pop up asking for a belt cleaning
	gMachine.St.CleaningBelt.xCleanRequired := (tiSumTimeToCleanBelt>=gMachine.parSw.CleanBelt.tiCleaningBeltByTime) AND
												enCleanBeltUvStep=CLN_BELT_READY_TO_CLEAN AND
												xReadyToCleanBelt AND
												gMachine.parSw.CleanBelt.xCleanBeltByTime;

	//If the belt is not running, it is not possible to clean it
	IF NOT gBelt.states.xRuningBelt THEN
		gMachine.commands.CleanBelt.xCleanBeltResetRelay := gMachine.AutoCmd.xReset AND gMachine.In.CleanBelt.xError;
		gMachine.commands.CleanBelt := ResetCleanBeltCommands;
		xCleanBeltOrder := FALSE;
		RETURN;
	END_IF

	//////////////////////
	// OUTPUT management
	//////////////////////
	//Clean belt
	xEnableCleanBeltMotorMovement := 	NOT gMachine.In.CleanBelt.xOpenGuide AND
										gMachine.In.CleanBelt.xHighPosition AND
										NOT tp_ToSwapCleanBeltMtrDirection.Q;

	//Pneumatic
	gMachine.commands.CleanBelt.xPistonFlojet := 	tofCleaningTrayBelt.Q AND
													NOT gMachine.In.CleanBelt.xOpenGuide AND
													gMachine.St.CleaningBelt.xCleaningProcessOnGoing;

	//Motor
	tp_ToSwapCleanBeltMtrDirection.IN:= EDGEPOS(xCleanBeltMoveFwd) OR EDGEPOS(xCleanBeltMoveBwd);
	tp_ToSwapCleanBeltMtrDirection.PT := gMachine.St.CleaningBelt.TimeDelaySwapDirBeltCleanMotor := t#2s;
	tp_ToSwapCleanBeltMtrDirection();

	gMachine.commands.CleanBelt.xCleanBeltMoveFwd := 	xCleanBeltMoveFwd AND
														xEnableCleanBeltMotorMovement;

	gMachine.commands.CleanBelt.xCleanBeltMoveBwd := 	xCleanBeltMoveBwd AND
														xEnableCleanBeltMotorMovement;

END_ACTION
```

#### CleanBeltWater.st
```iecst
ACTION CleanBeltWater:

	//To review if gBeltClean package will be used without line

	gBeltClean.Parameters.Mode := gMachine.St.Mode;
	gBeltClean.Parameters.rBeltSpeed := gBelt.states.rCurrentSpeed;
	gBeltClean.Parameters.xBeltRunning := gBelt.states.xRuningBelt;
	gBeltClean.Parameters.xBeltEmpty := gThicknessCtrl.status.Belt.xBeltEmpty;
	gMachine.St.CleaningBelt.xCleaningProcessOnGoing := gBeltClean.Status.xCleaning;
	IF gMachine.commands.CleanBelt.xStart AND gBeltClean.Status.xCleanRequested THEN
		gBeltClean.Commands.xAcceptRequest := TRUE;
	END_IF
	gBeltClean.Inputs.xEnteringMedia := EDGEPOS (gMachine.St.ProductDetect.xProductDetectL1);
	gBeltClean.Commands.xMute := gMachine.AutoCmd.xMuteAlarms;
	gBeltClean.Commands.xReset := gMachine.AutoCmd.xReset;
	gMachine.commands.CleanBelt := ResetCleanBeltCommands;
	gMachine.parSw.CleanBelt.iBeltSpeed := REAL_TO_UINT(gBeltClean.ParSw.rCleanBeltSpeed);

	//outputs
	gMachine.commands.CleanBelt.xPistonFlojet := gBeltClean.Outputs.xRiseCleaningSystem;
	gMachine.commands.CleanBelt.xCleanBeltPump := gBeltClean.Outputs.xPumpOn;
	//gBeltClean.Outputs.xAirTurbineOn Directly on Outputs
	//gBeltClean.Outputs.xAirTurbineVSDReset Directly on Outputs

END_ACTION
```

#### CleanSystem.st
```iecst
ACTION CleanSystem:

	//Variable used for all the counters of time. Counting seconds
	xEdge1sec := EDGEPOS(gPLC.xBlk_500ms);

	////////////////////////////////////////////////////////////////
	// Cleanning in Stop Mode
	// It doesnt work with delay and gap time
	////////////////////////////////////////////////////////////////

	IF gMachine.parSw.Clean.xEnableCleaningInStopMode AND gMachine.St.AutoMode.xStop AND xEdge1sec THEN
		uiSecondsToCleanStop := UDINT_SUB(uiSecondsToCleanStop, 1); // Value assigned after a cleaning
	END_IF
	IF EDGEPOS(uiSecondsToCleanStop = 0)  THEN
		gMachine.AutoCmd.xCleanningByTimeInStopMode:= TRUE;
	END_IF

	//Time for the next cleaning //Write 0 minutes to clean if cleaning is not activated
	IF gMachine.parSw.Clean.xEnableCleaningInStopMode THEN
		IF tiPrevToCleanWhenPrinterStopped<>gMachine.parSw.Clean.tiToCleanWhenPrinterStopped THEN
			tiPrevToCleanWhenPrinterStopped := gMachine.parSw.Clean.tiToCleanWhenPrinterStopped;
			uiSecondsToCleanStop := TIME_TO_UDINT(MAX(gMachine.parSw.Clean.tiToCleanWhenPrinterStopped, MIN_CLEANING_STOPPED)) / 1000;
		END_IF
		gMachine.St.Cleaning.MinutesInStopForClean := uiSecondsToCleanStop / 60;
	ELSE
		gMachine.St.Cleaning.MinutesInStopForClean := 0;
	END_IF

	////////////////////////////////
	// Cleaning By pieces
	////////////////////////////////

	IF gMachine.parSw.Clean.xCleanSystemByPieces THEN

		// Line 1
		IF  EDGEPOS (gMachine.St.ProductDetect.xProductDetectL1) AND gMachine.St.Position.xInPrint THEN
			gMachine.St.Cleaning.iPieceCounterBtwCleaningsL1:= gMachine.St.Cleaning.iPieceCounterBtwCleaningsL1+1;
		END_IF

		//Reset counter when setpoint is changed
		IF iPrevPiecesNumberToCleanL1<>gMachine.parSw.Clean.iPiecesNumberToCleanL1 THEN
			iPrevPiecesNumberToCleanL1 := gMachine.parSw.Clean.iPiecesNumberToCleanL1;
			gMachine.St.Cleaning.iPieceCounterBtwCleaningsL1:=0;
		END_IF

		//Reset counter L1
		IF gMachine.St.Cleaning.iPieceCounterBtwCleaningsL1 >= gMachine.parSw.Clean.iPiecesNumberToCleanL1 THEN
			gMachine.AutoCmd.xCleanningByPiecesL1:=TRUE; //Reset once machine is cleaning
			gMachine.St.Cleaning.iPieceCounterBtwCleaningsL1:=0;
		END_IF

		// Line 2
		IF  EDGEPOS (gMachine.St.ProductDetect.xProductDetectL2) AND gMachine.St.Position.xInPrint THEN
			gMachine.St.Cleaning.iPieceCounterBtwCleaningsL2:= gMachine.St.Cleaning.iPieceCounterBtwCleaningsL2+1;
		END_IF

		//Reset counter when setpoint is changed
		IF iPrevPiecesNumberToCleanL2<>gMachine.parSw.Clean.iPiecesNumberToCleanL2 THEN
			iPrevPiecesNumberToCleanL2 := gMachine.parSw.Clean.iPiecesNumberToCleanL2;
			gMachine.St.Cleaning.iPieceCounterBtwCleaningsL2:=0;
		END_IF

		//Reset counter L2
		IF gMachine.St.Cleaning.iPieceCounterBtwCleaningsL2 >= gMachine.parSw.Clean.iPiecesNumberToCleanL2 THEN
			gMachine.AutoCmd.xCleanningByPiecesL2:=TRUE; //Reset once machine is cleaning
			gMachine.St.Cleaning.iPieceCounterBtwCleaningsL2:=0;
		END_IF

	ELSE
		gMachine.St.Cleaning.iPieceCounterBtwCleaningsL1:=0;
		gMachine.St.Cleaning.iPieceCounterBtwCleaningsL2:=0;
	END_IF

	////////////////////////////////
	//	Cleanning Blocks by time
	////////////////////////////////

	IF gMachine.parSw.Clean.xCleanSystemByTime AND gMachine.St.AutoMode.xProduction AND xEdge1sec THEN
		uiSecondsToCleanProd := UDINT_SUB(uiSecondsToCleanProd, 1); // Value assigned after a cleaning
	END_IF
	IF EDGEPOS(uiSecondsToCleanProd = 0)  THEN
		gMachine.AutoCmd.xCleanningByTimeProd := TRUE;
	END_IF

	IF gMachine.parSw.Clean.xCleanSystemByTime THEN
		IF tiPrevCleaningByTime<>gMachine.parSw.Clean.tiCleaningByTime THEN
			tiPrevCleaningByTime := gMachine.parSw.Clean.tiCleaningByTime;
			uiSecondsToCleanProd := TIME_TO_UDINT(MAX(gMachine.parSw.Clean.tiCleaningByTime, MIN_CLEANING_BY_TIME)) / 1000;
		END_IF
		gMachine.St.Cleaning.MinutesInProdForClean := uiSecondsToCleanProd / 60;
	ELSE
		gMachine.St.Cleaning.MinutesInProdForClean := 0;
	END_IF

	gMachine.St.Cleaning.MinutesForClean := MIN(gMachine.St.Cleaning.MinutesInStopForClean, gMachine.St.Cleaning.MinutesInProdForClean);

	////////////////////////////////////////////////////////////////
	// Cleaning By External Order
	// gMachine.In.xExternalCleaningOrder in Mapping Inputs
	////////////////////////////////////////////////////////////////

	// Reference Jira  CRETALEGO-867: Cleaning system for signal external it isn't active only pulse.
	// It is solved adding an event by edge and setting this timer to start external cleaning order
	// Safety for order external, it is just executed when Printer is in cap or production

	// Timer management
	T_ExternalCleaningOrder.IN:= gMachine.In.xExternalCleaningOrder AND (gMachine.St.Cleaning.enCleaningState = CLN_NOT_CLEANING) AND gMachine.St.Mode.xAuto;
	T_ExternalCleaningOrder.PT:= T#500ms;
	T_ExternalCleaningOrder();
	IF EDGEPOS(T_ExternalCleaningOrder.Q) THEN
		gMachine.AutoCmd.xCleanningByExtOrder := TRUE;
	END_IF

	////////////////////////////////
	//	Cleaning while Time NOT Cleaned whatever the state
	////////////////////////////////
	IF gMachine.Pt.Clean.xEnabledCleanTotalTime AND xEdge1sec THEN
		uiSecondsToCleanTotal := UDINT_SUB(uiSecondsToCleanTotal, 1); // Value assigned after a cleaning
	END_IF
	IF EDGEPOS(uiSecondsToCleanTotal = 0 AND gMachine.St.Mode.xAuto AND gMachine.Pt.Clean.xEnabledCleanTotalTime)  THEN
		gMachine.AutoCmd.xCleanningByTotalTime:= TRUE;
	END_IF

	//Time for the next cleaning //Write 0 minutes to clean if cleaning is not activated
	IF gMachine.Pt.Clean.xEnabledCleanTotalTime THEN
		gMachine.St.Cleaning.MinutesTotalTimeForClean := uiSecondsToCleanTotal / 60;
	ELSE
		gMachine.St.Cleaning.MinutesTotalTimeForClean := 0;
	END_IF

	// Preparing gap in line (Add here all cleaning orders)
	IF gMachine.AutoCmd.xCleanningByExtOrder OR
		gMachine.AutoCmd.xCleanningByPiecesL1 OR
		gMachine.AutoCmd.xCleanningByPiecesL2 OR
		gMachine.AutoCmd.xCleanningByTimeProd OR
		gMachine.AutoCmd.xCleanningByTotalTime THEN

		IF gMachine.Pt.xControlledByLine THEN
			gMachine.St.Cleaning.xCleanRequestToLine := TRUE;

		ELSIF gMachine.Pt.xControlledRemotely THEN
			tonWaitToCleanRemote.IN := TRUE;
			tonWaitToCleanRemote.PT := T#10m;
			tonWaitToCleanRemote();
			gMachine.St.Cleaning.xCleanRequired := TRUE;
			gMachine.St.Cleaning.xCleanInminent := tonWaitToCleanRemote.ET > (tonWaitToCleanRemote.PT - T#30s); // Activate 30" before final activation
			IF tonWaitToCleanRemote.Q THEN
				gMachine.commands.xClean:=TRUE;
				tonWaitToCleanRemote(IN := FALSE); //Reset de remote timer
			END_IF

		ELSE
			gMachine.commands.xClean:=TRUE;

		END_IF
	END_IF

	// Delay control function
	FbCleanDelayControl_1.Start:= xOrderToGap;
	FbCleanDelayControl_1.T_delay_L1:= gMachine.parSw.Clean.tiTimeDelayToCleanL1;
	FbCleanDelayControl_1.T_delay_L2:= gMachine.parSw.Clean.tiTimeDelayToCleanL2;
	FbCleanDelayControl_1.Doble:= gMachine.parSw.Dtp.xDoubleLine;
	FbCleanDelayControl_1.t_Gap:= gMachine.parSw.Clean.tiTimeDelayGapToClean;
	FbCleanDelayControl_1();

	xDelayCleaningOk:= FbCleanDelayControl_1.End; //This signal allow start cleaning, the gap is and delay line are properly executed.

	// Mapping outputs to start getting gap in Lines
	gMachine.Out.xLine1ReadyToClean:= FbCleanDelayControl_1.Out_L1;
	gMachine.Out.xLine2ReadyToClean:= FbCleanDelayControl_1.Out_L2;

	////////////////////////////////////////////////////////////////
	// Cleaning blocks togheter or separate
	////////////////////////////////////////////////////////////////

	// A small state machine should be implemented here....
	//
	// Take care with action ControlState.st in Block Program !!!!
	//
	// Initial system cleaning
	// Configure first block
	// Prepare for next
	// Start next block
	// Finshed lastest block
	//
	// Enabled blocks for cleaning at once or at same time

	//Remove pending cleanings if not in Auto Mode
	IF NOT gMachine.St.Mode.xAuto THEN
		enCleaningState := CLN_NOT_CLEANING;
		ResetCleanOrders;
	END_IF

	CASE enCleaningState OF

		CLN_NOT_CLEANING:
			//Be ready to detect when each block has finished
			FOR iIndexBlock:=GC_FIRST_BLOCK TO gMachine.Pt.CT.iNumBlocks DO
				arBlockCleaningEnded[iIndexBlock]:=FALSE;
				gBlock[iIndexBlock].commands.xStartToCleanOrder:= FALSE;
			END_FOR
			IF NOT gMachine.Pt.xControlledByLine THEN gMachine.St.xBeltRunPrevToClean := gBelt.states.xRuningBelt; END_IF

			//Cleaning with delay
			IF (gMachine.commands.xClean AND NOT gMachine.St.Position.xInCap AND NOT gMachine.St.AutoMode.xLaboratory) OR
				gBlock[1].commands.xForceCleanDelay OR
				gBlock[2].commands.xForceCleanDelay THEN

				enCleaningState:= CLN_LINEDELAYING_GAP;
			END_IF

			//Cleaning without Delay
			IF ((gMachine.AutoCmd.xCleanningByTimeInStopMode OR gMachine.commands.xClean OR gMachine.AutoCmd.xCleanningByExtOrder) AND
				(gMachine.St.Position.xInCap OR gMachine.St.AutoMode.xLaboratory)) OR
				gBlock[1].commands.xForceCleanNoDelay OR
				gBlock[2].commands.xForceCleanNoDelay THEN

				enCleaningState:= CLN_READY_TO_CLEAN;

			END_IF
			xCleanSequencially:=FALSE;
			xOrderToGap:=FALSE;

		CLN_LINEDELAYING_GAP:
			xOrderToGap:=TRUE;
			IF xDelayCleaningOk THEN
				enCleaningState:= CLN_READY_TO_CLEAN;
			END_IF

		CLN_READY_TO_CLEAN:
			IF gBlock[1].commands.xForceCleanDelay OR gBlock[1].commands.xForceCleanNoDelay THEN
				enCleaningState:= CLN_CLEANING_JUST1_START;

			ELSIF gBlock[2].commands.xForceCleanDelay OR gBlock[2].commands.xForceCleanNoDelay THEN
				enCleaningState:= CLN_CLEANING_JUST2_START;

			ELSIF gMachine.parSw.Clean.xCleaningBlocksInSeq THEN
				enCleaningState:= CLN_CLEANING_1_START;

			ELSE
				enCleaningState:= CLN_CLEANING_ALL_START;

			END_IF
			ResetCleanOrders;

		CLN_CLEANING_ALL_START:
			// There is one printer command joined for all blocks
			xAllBlocksCleaning:=TRUE;
			FOR iIndexBlock:=GC_FIRST_BLOCK TO gMachine.Pt.CT.iNumBlocks DO

				//Check if the command is edge or not
				iReasonToSendCleanOrder.0 := gBlock[iIndexBlock].Status.PositionState<>BLOCKP_CLEANING;
				iReasonToSendCleanOrder.1 := gBlock[iIndexBlock].Status.xEnabledToClean;
				iReasonToSendCleanOrder.2 := gBlock[iIndexBlock].Status.xEnabledMovements;

				//Sent the order if not sended and the block is able to clean
				IF iReasonToSendCleanOrder = 2#0111 THEN
					gBlock[iIndexBlock].commands.xStartToCleanOrder:= TRUE;
					xAllBlocksCleaning:=FALSE; //If any block not cleaning, fall the signal
				END_IF

			END_FOR

			//To be sure that the order has been sent and not resent it again
			IF xAllBlocksCleaning THEN
				enCleaningState:= CLN_CLEANING_ALL_CLEANING;
			END_IF

		CLN_CLEANING_ALL_CLEANING:
			//Check if ALL Blocks have finished
			xAllBlocksCleaningEnded:=TRUE;
			FOR iIndexBlock:=GC_FIRST_BLOCK TO gMachine.Pt.CT.iNumBlocks DO
				IF NOT gBlock[iIndexBlock].Status.xCleaningDone THEN
					xAllBlocksCleaningEnded:=FALSE;
				END_IF
			END_FOR

			IF xAllBlocksCleaningEnded THEN
				enCleaningState:= CLN_NOT_CLEANING; // Cleaning state in block finished
				ResetCleanOrders;
				ResetCleanCountersAndTimers;
			END_IF

		CLN_CLEANING_1_START:
			xCleanSequencially:=TRUE;
			iIndexBlock:=1;
			CleanBlockStart;

		CLN_CLEANING_1_CLEANING:
			iIndexBlock:=1;
			CleanBlockCleaning;

		CLN_CLEANING_BTW_BLOCKS:
			//Timer management for cleaning between blocks
			T_BtwnCleans.IN:= TRUE;
			T_BtwnCleans.PT:= gMachine.parSw.Clean.tiBetweenCleaningBlocks;
			T_BtwnCleans();
			IF T_BtwnCleans.Q THEN
				enCleaningState:= CLN_CLEANING_2_START;
				T_BtwnCleans.IN:= FALSE;
				T_BtwnCleans(); //This is to fall the output of the Timer and be able to count on next cycle
			END_IF

		CLN_CLEANING_2_START:
			iIndexBlock:=2;
			CleanBlockStart;

		CLN_CLEANING_2_CLEANING:
			iIndexBlock:=2;
			CleanBlockCleaning;

		CLN_CLEANING_JUST1_START:
			iIndexBlock:=1;
			CleanBlockStart;

		CLN_CLEANING_JUST1_CLEANING:
			iIndexBlock:=1;
			CleanBlockCleaning;

		CLN_CLEANING_JUST2_START:
			iIndexBlock:=2;
			CleanBlockStart;

		CLN_CLEANING_JUST2_CLEANING:
			iIndexBlock:=2;
			CleanBlockCleaning;

	END_CASE

	gMachine.St.Cleaning.enCleaningState := enCleaningState;
	//Return value to Sw
	CASE enCleaningState OF
		CLN_NOT_CLEANING: gMachine.St.Cleaning.iCleaningState := 1;
		CLN_LINEDELAYING_GAP: gMachine.St.Cleaning.iCleaningState := 2;
		CLN_READY_TO_CLEAN: gMachine.St.Cleaning.iCleaningState := 3;
		CLN_CLEANING_ALL_START: gMachine.St.Cleaning.iCleaningState := 4;
		CLN_CLEANING_ALL_CLEANING: gMachine.St.Cleaning.iCleaningState := 5;
		CLN_CLEANING_1_START: gMachine.St.Cleaning.iCleaningState := 6;
		CLN_CLEANING_1_CLEANING: gMachine.St.Cleaning.iCleaningState := 7;
		CLN_CLEANING_BTW_BLOCKS: gMachine.St.Cleaning.iCleaningState := 8;
		CLN_CLEANING_2_START: gMachine.St.Cleaning.iCleaningState := 9;
		CLN_CLEANING_2_CLEANING: gMachine.St.Cleaning.iCleaningState := 10;
		CLN_CLEANING_JUST1_START: gMachine.St.Cleaning.iCleaningState := 11;
		CLN_CLEANING_JUST1_CLEANING: gMachine.St.Cleaning.iCleaningState := 12;
		CLN_CLEANING_JUST2_START: gMachine.St.Cleaning.iCleaningState := 13;
		CLN_CLEANING_JUST2_CLEANING: gMachine.St.Cleaning.iCleaningState := 14;
	END_CASE
END_ACTION

ACTION CleanBlockStart:

	iReasonToSendCleanOrder.0 := gBlock[iIndexBlock].Status.PositionState<>BLOCKP_CLEANING;
	iReasonToSendCleanOrder.1 := gBlock[iIndexBlock].Status.xEnabledToClean;
	iReasonToSendCleanOrder.2 := gBlock[iIndexBlock].Status.xEnabledMovements;

	//Sent the order if not sended and the block is able to clean
	IF iReasonToSendCleanOrder = 2#0111 THEN
			gBlock[iIndexBlock].commands.xStartToCleanOrder:= TRUE;

	//If cleaning or not possible to clean, go to next step
	ELSE
		gBlock[iIndexBlock].commands.xStartToCleanOrder:= FALSE;
		IF xCleanSequencially THEN
			CASE iIndexBlock OF
				1:	enCleaningState:= CLN_CLEANING_1_CLEANING;
				2:	enCleaningState:= CLN_CLEANING_2_CLEANING;
			END_CASE
		ELSE
			CASE iIndexBlock OF
				1:	enCleaningState:= CLN_CLEANING_JUST1_CLEANING;
				2:	enCleaningState:= CLN_CLEANING_JUST2_CLEANING;
			END_CASE
		END_IF
	END_IF

END_ACTION

ACTION CleanBlockCleaning:

	//Check if ALL Blocks have finished
	IF gBlock[iIndexBlock].Status.xCleaningDone THEN
		IF xCleanSequencially THEN
			CASE iIndexBlock OF
				1:	enCleaningState:= CLN_CLEANING_BTW_BLOCKS;
				2:	enCleaningState:= CLN_NOT_CLEANING; ResetCleanOrders;
			END_CASE
		ELSE
			enCleaningState:= CLN_NOT_CLEANING;
			ResetCleanOrders; // Cleaning state in block finished
			ResetCleanCountersAndTimers;
		END_IF
	END_IF

END_ACTION

ACTION ResetCleanOrders:

	//Reset Cleaning orders once the machine is cleaning
	gMachine.AutoCmd.xCleanningByTimeProd:=FALSE;
	gMachine.AutoCmd.xCleanningByTotalTime:=FALSE;
	gMachine.AutoCmd.xCleanningByExtOrder:=FALSE;
	gMachine.AutoCmd.xCleanningByPiecesL1:=FALSE;
	gMachine.AutoCmd.xCleanningByPiecesL2:=FALSE;
	gMachine.AutoCmd.xCleanningByTimeInStopMode:=FALSE;
	gBlock[1].commands.xForceCleanNoDelay:=FALSE;
	gBlock[2].commands.xForceCleanNoDelay:=FALSE;
	gBlock[1].commands.xForceCleanDelay:= FALSE;
	gBlock[2].commands.xForceCleanDelay:=FALSE;
	gMachine.St.Cleaning.xCleanRequestToLine := FALSE;
	gMachine.commands.xClean := FALSE;
	gMachine.St.Cleaning.xCleanRequired := FALSE;
	gMachine.St.Cleaning.xCleanInminent := FALSE;
	tonWaitToCleanRemote(IN := FALSE); //Reset de remote timer

END_ACTION

ACTION ResetCleanCountersAndTimers:

	iSecondsNoCleaned := 0;

	uiSecondsToCleanStop := TIME_TO_UDINT(MAX(gMachine.parSw.Clean.tiToCleanWhenPrinterStopped, MIN_CLEANING_STOPPED)) / 1000;
	uiSecondsToCleanProd := TIME_TO_UDINT(MAX(gMachine.parSw.Clean.tiCleaningByTime, MIN_CLEANING_BY_TIME)) / 1000;
	uiSecondsToCleanTotal := 24 * 3600; // Maximum 1 day

END_ACTION
```

#### JamSensors.st
```iecst
ACTION JamSensors:

	IF NOT gMachine.parSw.xJamDetectEnable THEN
		RETURN;
	END_IF

	FOR iIndexInks :=1 TO MAX_LAST_INK DO
		gJamPerInk[iIndexInks].xAlrJamCrash	:= gJamDetect[gJamPerInk[iIndexInks].iJamDevice].Alarms.xAlrJamCrash[gJamPerInk[iIndexInks].iJamSensor];
		gJamPerInk[iIndexInks].xAlrJamTest	:= gJamDetect[gJamPerInk[iIndexInks].iJamDevice].Alarms.xAlrJamTest[gJamPerInk[iIndexInks].iJamSensor];
		gJamPerInk[iIndexInks].xAlrLowJamCrash	:= gJamDetect[gJamPerInk[iIndexInks].iJamDevice].Alarms.xAlrJamLowCrash;
	END_FOR

	FOR iIndexCuringLedLamps :=1 TO MAX_LAST_CURING_LED DO
		gJamPerCuringLed[iIndexCuringLedLamps].xAlrJamCrash	:= gJamDetect[gJamPerCuringLed[iIndexCuringLedLamps].iJamDevice].Alarms.xAlrJamCrash[gJamPerCuringLed[iIndexCuringLedLamps].iJamSensor];
		gJamPerCuringLed[iIndexCuringLedLamps].xAlrJamTest	:= gJamDetect[gJamPerCuringLed[iIndexCuringLedLamps].iJamDevice].Alarms.xAlrJamTest[gJamPerCuringLed[iIndexCuringLedLamps].iJamSensor];
		gJamPerCuringLed[iIndexCuringLedLamps].xAlrLowJamCrash	:= gJamDetect[gJamPerCuringLed[iIndexCuringLedLamps].iJamDevice].Alarms.xAlrJamLowCrash;
	END_FOR

	gJamCamera.xAlrJamCrash	:= gJamDetect[gJamCamera.iJamDevice].Alarms.xAlrJamCrash[gJamCamera.iJamSensor];
	gJamCamera.xAlrJamTest	:= gJamDetect[gJamCamera.iJamDevice].Alarms.xAlrJamTest[gJamCamera.iJamSensor];
	gJamCamera.xAlrLowJamCrash := gJamDetect[gJamCamera.iJamDevice].Alarms.xAlrJamLowCrash;

END_ACTION
```

#### LightBeacon.st
```iecst
ACTION LightBeacon:

	// Green: Started and not any alarm
	gMachine.Out.xGreenLight:= 	gBelt.states.xRuningBelt OR
								(NOT gBelt.states.xRuningBelt AND gMachine.St.AutoMode.xPause AND gPLC.xBlk_500ms);

	// Red: Started and critical alarm
	gMachine.Out.xRedLight:= 	gMachine.AlSummary.xAlarmCritical OR
								(gMachine.AlSummary.xAlarmStop AND gPLC.xBlk_500ms) OR
								(xAnyInkCriticalAlrm AND gPLC.xBlk_2s);

	// Yellow: Started and stop alarm
	gMachine.Out.xYellowLight:= gMachine.AlSummary.xAnyWarning;

	////////////////////////////
	// LIGHT RESET
	////////////////////////////
	gMachine.Out.xLightReset:= gMachine.AutoCmd.xReset;

END_ACTION

ACTION RgbLigths:

	//As just one color may be activated at the same time, we need to priorize color code
	ResetRgbColors;
	IF gSafetyController.Inputs.xPrinterMaintenanceKey THEN
		xRedLight := gPLC.xBlk_200ms;
	ELSIF gSafetyController.Alarms.xCriticalAlarm THEN
		xRedLight := TRUE;
	ELSIF gMachine.AlSummary.xAlarmCritical OR gMachine.AlSummary.xAlarmStop THEN
		xYellowLight := gPLC.xBlk_1s;
	ELSIF gMachine.St.Mode.xAuto THEN
		xWhiteLight:= gMachine.St.Mode.xAuto;
	ELSIF gMachine.AlSummary.xAnyWarning THEN
		xYellowLight := TRUE;
	END_IF

	//Conversion to RGB
	gMachine.Out.xGreenLight := xYellowLight OR xGreenLight;
	gMachine.Out.xRedLight := xYellowLight OR xRedLight;
	gMachine.Out.xBlueLight := xBlueLight;
	gMachine.Out.xWhiteLight := xWhiteLight;

END_ACTION

ACTION ResetRgbColors:
	xGreenLight := FALSE;
	xRedLight := FALSE;
	xBlueLight := FALSE;
	xWhiteLight := FALSE;
	xYellowLight := FALSE;
END_ACTION
```

#### PowerCtrl.st
```iecst
ACTION PowerCtrl:

	// If alarm Sai PowerOff and Keep Pcs Cms
	T_OnPcs.IN:= NOT gMachine.Al.Alarm.xAlarmSAIPowerOff;
	T_OnPcs.PT:= T#5S;
	T_OnPcs();

	xOnPcs:= T_OnPcs.Q AND gMachine.parSw.PCs.xKeepPcsOn;

	// Starting PC1
	T_WaitPC1.IN:= xOnPcs AND NOT gMachine.In.xPC1Ok AND NOT T_OnPC1.Q;
	T_WaitPC1.PT:= T#3S;
	T_WaitPC1();

	T_OnPC1.IN:=T_WaitPC1.Q;
	T_OnPC1.PT:= T#500MS;
	T_OnPC1();

	gMachine.Out.xPC1Start:= T_WaitPC1.Q;

	// Starting PC2
	T_WaitPC2.IN:= xOnPcs AND NOT gMachine.In.xPC2Ok AND NOT T_OnPC2.Q;
	T_WaitPC2.PT:= T#3S;
	T_WaitPC2();

	T_OnPC2.IN:=T_WaitPC2.Q;
	T_OnPC2.PT:= T#500MS;
	T_OnPC2();

	gMachine.Out.xPC2Start:= T_WaitPC2.Q;

END_ACTION
```

#### ProgramsManager.st
```iecst
ACTION ProgramsManager:

	// This functionality is currently disabled
	RETURN;

	IF EDGEPOS(gMachine.Pt.ConfigNameID<>0) THEN
		AssignProgramIdentification;

		iSuspendInit := ST_tmp_suspend(identInitialize);
	END_IF

	//Manage Analog thickness execution
	IF EDGEPOS(gDing.Parameters.xDingInstalled AND NOT gPLC.xFirst_Scan) THEN

		AssignProgramIdentification;
		iResumeAnalogFast := ST_tmp_resume(identAnalogFast);
		AssignProgramIdentification;
		iResumeAnalogThick := ST_tmp_resume(identAnalogThick);

		nResumeAnalog := nResumeAnalog + 1;
	END_IF
	IF EDGEPOS(gPhotoCells.status.xInstalled AND NOT gDing.State.xDingInstalled AND NOT gPLC.xFirst_Scan) THEN

		AssignProgramIdentification;
		iSuspendAnalogFast := ST_tmp_suspend(identAnalogFast);
		AssignProgramIdentification;
		iSuspendAnalogThick := ST_tmp_suspend(identAnalogThick);

		nSuspendAnalog := nSuspendAnalog + 1;
	END_IF

	IF EDGEPOS(gPhotoCells.parameters.xInstall AND NOT gPLC.xFirst_Scan) THEN
		ResetResumeLaserResult;

		//In simulation this is not running
		IF gMachine.St.HwData.Family <> FAMILY_BRAUTOMATIONRUNTIME THEN
			AssignProgramIdentification;
			iResumeStepper2 := ST_tmp_resume(identStepper2);
			AssignProgramIdentification;
			iResumeStepper1 := ST_tmp_resume(identStepper1);
			AssignProgramIdentification;
			iResumeInitStepper := ST_tmp_resume(identInitStepper);
		END_IF
		AssignProgramIdentification;
		iResumeLaserFast := ST_tmp_resume(identLaserFast);
		AssignProgramIdentification;
		iResumeLaserCtrl := ST_tmp_resume(identLaserCtrl);
		CASE gMachine.Pt.MachineModel OF
			Type_P4_12B,
			Type_P4_12B_L,
			Type_P4_6B,
			Type_P4_CBK,
			Type_P4_6B_L:
				AssignProgramIdentification;
				iResumeAxisStepper1 := ST_tmp_resume(identAxisStepper1);
				AssignProgramIdentification;
				iResumeAxisStepper2 := ST_tmp_resume(identAxisStepper2);
		END_CASE
		nResumeLaser := nResumeLaser + 1;
	END_IF
	IF EDGEPOS(gDing.State.xDingInstalled AND NOT gPhotoCells.status.xInstalled AND NOT gPLC.xFirst_Scan) THEN
		ResetSuspendLaserResult;

		//In simulation this is not running
		IF gMachine.St.HwData.Family <> FAMILY_BRAUTOMATIONRUNTIME THEN
			AssignProgramIdentification;
			iSuspendStepper2 := ST_tmp_suspend(identStepper2);
			AssignProgramIdentification;
			iSuspendStepper1 := ST_tmp_suspend(identStepper1);
			AssignProgramIdentification;
			iSuspendInitStepper := ST_tmp_suspend(identInitStepper);
			AssignProgramIdentification;
		END_IF
		iSuspendLaserFast := ST_tmp_suspend(identLaserFast);
		AssignProgramIdentification;
		iSuspendLaserCtrl := ST_tmp_suspend(identLaserCtrl);
		CASE gMachine.Pt.MachineModel OF
			Type_P4_12B,
			Type_P4_12B_L,
			Type_P4_6B,
			Type_P4_CBK,
			Type_P4_6B_L:
				AssignProgramIdentification;
				iSuspendAxisStepper1 := ST_tmp_suspend(identAxisStepper1);
				AssignProgramIdentification;
				iSuspendAxisStepper2 := ST_tmp_suspend(identAxisStepper2);
		END_CASE
		nSuspendLaser := nSuspendLaser + 1;
	END_IF

	nProgramManager := nProgramManager + 1;
END_ACTION

ACTION ResetSuspendLaserResult:
	iSuspendStepper2 := 10;
	iSuspendStepper1 := 10;
	iSuspendInitStepper := 10;
	iSuspendLaserFast := 10;
	iSuspendLaserCtrl := 10;
	iSuspendAxisStepper1 := 10;
	iSuspendAxisStepper2 := 10;
END_ACTION

ACTION ResetResumeLaserResult:
	iResumeStepper2 := 10;
	iResumeStepper1 := 10;
	iResumeInitStepper := 10;
	iResumeLaserFast := 10;
	iResumeLaserCtrl := 10;
	iResumeAxisStepper1 := 10;
	iResumeAxisStepper2 := 10;
END_ACTION

ACTION AssignProgramIdentification:

	//Determine identificator for programs to allow working with them
	iGroup := 0; //Currently not used
	stProgramName := 'Initialize';
	ST_ident(ADR(stProgramName),iGroup,ADR(identInitialize));

	stProgramName := 'Analog_Fas';
	ST_ident(ADR(stProgramName),iGroup,ADR(identAnalogFast));
	stProgramName := 'AnalogThic';
	ST_ident(ADR(stProgramName),iGroup,ADR(identAnalogThick));

	stProgramName := 'InitSteprs';
	ST_ident(ADR(stProgramName),iGroup,ADR(identInitStepper));
	stProgramName := 'Stepper3L1';
	ST_ident(ADR(stProgramName),iGroup,ADR(identStepper1));
	stProgramName := 'Stepper3L2';
	ST_ident(ADR(stProgramName),iGroup,ADR(identStepper2));
	stProgramName := 'Stepper3L';
	ST_ident(ADR(stProgramName),iGroup,ADR(identAxisStepper1));
	stProgramName := 'Gear3L';
	ST_ident(ADR(stProgramName),iGroup,ADR(identAxisStepper2));
	stProgramName := 'nSens_Fast';
	ST_ident(ADR(stProgramName),iGroup,ADR(identLaserFast));
	stProgramName := 'nSensorCtr';
	ST_ident(ADR(stProgramName),iGroup,ADR(identLaserCtrl));

END_ACTION
```

#### ResetRouterAndCB.st
```iecst
ACTION ResetRouterAndCB:

	// Reset Router
	tof_ResetRouter.IN:=gMachine.commands.xResetRouter;
	tof_ResetRouter.PT:= T#6s;
	tof_ResetRouter();
	gMachine.commands.xResetRouter:= FALSE;

	gMachine.Out.xResetRouter:=tof_ResetRouter.Q;

	// Reset CB1/CB2 (Always together, just one button in interface)
	tof_ResetCB1.IN:=gMachine.commands.xResetCB;
	tof_ResetCB1.PT:= T#4s;
	tof_ResetCB1();
	gMachine.commands.xResetCB:= FALSE;

	gMachine.Out.xResetCB1:=tof_ResetCB1.Q;
	gMachine.Out.xResetCB2:=tof_ResetCB1.Q;

END_ACTION
```

#### SoundBeacon.st
```iecst
ACTION SoundBeacon:
	// Acoustic advise
	//
	// AutoReseteable Alarms sound management
	arNotLoadedImage	(xAlarm:= gMachine.Al.Warning.xNotLoadedImage OR gMachine.Al.Alarm.xNotLoadedImage, xSilence:=gMachine.AutoCmd.xMuteAlarms);
	arSAIFault			(xAlarm:= gMachine.Al.Warning.xSAIFault, xSilence:=gMachine.AutoCmd.xMuteAlarms);
	arBentTile			(xAlarm:= gMachine.Al.Warning.xBentTile, xSilence:=gMachine.AutoCmd.xMuteAlarms);
	arPDSensorErrorL1	(xAlarm:= gMachine.Al.Alarm.xPDBrokenSensorL1, xSilence:=gMachine.AutoCmd.xMuteAlarms);
	arPDSensorErrorL2	(xAlarm:= gMachine.Al.Alarm.xPDBrokenSensorL2, xSilence:=gMachine.AutoCmd.xMuteAlarms);
	arNoThicknessSystem	(xAlarm:= gMachine.Al.Alarm.xAlrThicknSystemNotSelected, xSilence:=gMachine.AutoCmd.xMuteAlarms);
	arSAIPowerFault		(xAlarm:= gMachine.Al.Alarm.xAlarmSAIPowerFault, xSilence:= gMachine.AutoCmd.xMuteAlarms);
	arHeaterTankPsu		(xAlarm:= gMachine.Al.Alarm.xHeaterTankPsu, xSilence:= gMachine.AutoCmd.xMuteAlarms);
	arAlrMountedPiece	(xAlarm:= gMachine.Al.Alarm.xAlarmMountedPiece, xSilence:= gMachine.AutoCmd.xMuteAlarms);
	arsWrongDingPos		(xAlarm:= gMachine.Al.Alarm.xAlrDingWrongPosition, xSilence:= gMachine.AutoCmd.xMuteAlarms);
	arsSwCriticalCondition(xAlarm:= gMachine.parSw.UI.xCriticalCondition, xSilence:= gMachine.AutoCmd.xMuteAlarms);
	arCommsPcPlc	(xAlarm:= gMachine.Al.Alarm.xAlarmComPcPLC, xSilence:=gMachine.AutoCmd.xMuteAlarms);

	//Stopped Media inside intermitent beep
	tpStoppedMediaInsd	(IN := gMachine.Al.Warning.xMediaStoppedInside, PT := T#3s);
	BlnkMediaInside		(xEnable := tpStoppedMediaInsd.Q, tTimeOn := T#100ms, tTimeOff := T#100ms);

	//Sound/Beep reasons
	//General
	reasonSoundGen.0 := arNotLoadedImage.xAlarmSound;
	reasonSoundGen.1 := arSAIFault.xAlarmSound;
	reasonSoundGen.2 := arBentTile.xAlarmSound;
	reasonSoundGen.3 := arNoThicknessSystem.xAlarmSound;
	reasonSoundGen.4 := arSAIPowerFault.xAlarmSound;
	reasonSoundGen.5 := arPDSensorErrorL1.xAlarmSound;
	reasonSoundGen.6 := arPDSensorErrorL2.xAlarmSound;
	reasonSoundGen.7 := arHeaterTankPsu.xAlarmSound;
	reasonSoundGen.8 := gBelt.AlSummary.xAlarmSound;
	reasonSoundGen.9 := gBlock[1].AlSummary.xAlarmSound;
	reasonSoundGen.10 := gBlock[2].AlSummary.xAlarmSound;
	reasonSoundGen.11 := gPhotoCells.AlSummary.xAlarmSound;
	reasonSoundGen.12 := gChiller[1].AlSummary.xAlarmSound;
	reasonSoundGen.13 := gChiller[2].AlSummary.xAlarmSound;
	reasonSoundGen.14 := gTransVacuum[1].AlSummary.xAlarmSound;
	reasonSoundGen.15 := gTransVacuum[2].AlSummary.xAlarmSound;
	reasonSoundGen.16 := gNonCrash[1].AlSummary.xAlarmSound;
	reasonSoundGen.17 := gNonCrash[2].AlSummary.xAlarmSound;
	reasonSoundGen.18 := gJamDetect[1].AlSummary.xAlarmSound;
	reasonSoundGen.19 := gJamDetect[2].AlSummary.xAlarmSound;
	reasonSoundGen.20 := gDing.AlSummary.xAlarmSound;
	reasonSoundGen.21 := arAlrMountedPiece.xAlarmSound;
	reasonSoundGen.22 := gCuringLed[iIndexWhiteCuringLedBar].AlSummary.xAlarmSound;
	reasonSoundGen.23 := gCuringLed[iIndexColorCuringLedBar].AlSummary.xAlarmSound;
	reasonSoundGen.24 := gPairedMotors[1].AlSummary.xAlarmSound;
	reasonSoundGen.25 := gPairedMotors[2].AlSummary.xAlarmSound;
	reasonSoundGen.26 := BlnkMediaInside.xOutput;
	reasonSoundGen.27 := arsWrongDingPos.xAlarmSound;
	reasonSoundGen.28 := arsSwCriticalCondition.xAlarmSound;

	reasonSoundGen2.0 := arCommsPcPlc.xAlarmSound;
	reasonSoundGen2.1 := gEdgeHoldDown.AlSummary.xAlarmSound;

	//Inks related reasons
	reasonSoundInks.0 := gInks[1].AlSummary.xAlarmSound;
	reasonSoundInks.1 := gInks[2].AlSummary.xAlarmSound;
	reasonSoundInks.2 := gInks[3].AlSummary.xAlarmSound;
	reasonSoundInks.3 := gInks[4].AlSummary.xAlarmSound;
	reasonSoundInks.4 := gInks[5].AlSummary.xAlarmSound;
	reasonSoundInks.5 := gInks[6].AlSummary.xAlarmSound;
	reasonSoundInks.6 := gInks[7].AlSummary.xAlarmSound;
	reasonSoundInks.7 := gInks[8].AlSummary.xAlarmSound;
	reasonSoundInks.8 := gInks[9].AlSummary.xAlarmSound;
	reasonSoundInks.9 := gInks[10].AlSummary.xAlarmSound;
	reasonSoundInks.10 := gInks[11].AlSummary.xAlarmSound;
	reasonSoundInks.11 := gInks[12].AlSummary.xAlarmSound;

	gMachine.Al.xAlarmSound:= (reasonSoundGen>0) OR (reasonSoundGen2>0) OR (reasonSoundInks>0);

	// Alarm sound output
	IF 	gMachine.AutoCmd.xMuteAlarms OR
		(gMachine.In.Buttons.xZero AND NOT (reasonSoundInks > 0) AND NOT gBlock[1].Al.xAlrSafetySystemInBlock) THEN

		gMachine.AlSummary.xAlarmSound:=FALSE;
	ELSE
		gMachine.AlSummary.xAlarmSound:= gMachine.Al.xAlarmSound;
	END_IF;

	SoundAtStart;

	//Buzzer management
	IF (iCountStartSound >= BEEP_START_COUNTS) THEN
		IF gBlock[1].Status.Motor.xBarsHoming OR
			gBlock[2].Status.Motor.xBarsHoming OR
			gBlock[1].Status.Icla.xHoming OR
			gBlock[2].Status.Icla.xHoming OR
			gEdgeHoldDown.status.xReferencing OR
			gPhotoCells.status.xReferencing THEN

			gMachine.Out.xBuzzerButtonPanel:=  gPLC.xBlk_1s;

		ELSIF gBelt.states.State = BELT_PREPARING_START THEN
			gMachine.Out.xBuzzerButtonPanel:=  gPLC.xBlk_500ms;

		ELSE
			gMachine.Out.xBuzzerButtonPanel:=  gMachine.AlSummary.xAlarmSound;
		END_IF

	ELSE
		gMachine.Out.xBuzzerButtonPanel:=  xStartSound;
	END_IF

END_ACTION

ACTION SoundAtStart:

	//Whit 5, we have 3 beeps at the begining
	IF iCountStartSound >= BEEP_START_COUNTS THEN
		RETURN;
	END_IF

	tonStartSound.IN := NOT tonStartSound.Q;
	tonStartSound.PT := t#1s;
	tonStartSound();

	IF EDGEPOS(tonStartSound.Q) THEN
		iCountStartSound := iCountStartSound + 1;
	END_IF

	xStartSound := (iCountStartSound MOD 2) = 0;

END_ACTION
```

#### Startup.st
```iecst
ACTION Startup:

	IF NOT gMachine.Pt.xAllowAutoStartUp OR NOT gMachine.parSw.xAutoStartEnabled THEN
		gMachine.St.StartUp.Status := STRUP_DISABLED;
		enStartUpStatus :=  STRUP_DISABLED;
		gMachine.St.StartUp.xReadyToAuto := TRUE;
		RETURN;
	END_IF

	IF (EDGENEG(gMachine.In.xSafetyEnabled) OR EDGENEG(gMachine.In.Buttons.xAuto)) AND
		(enStartUpStatus <> STRUP_CANCELLED OR  enStartUpStatus <> STRUP_READY OR enStartUpStatus <> STRUP_NOT_STARTED) THEN
			enStartUpStatus := STRUP_ERROR;
	END_IF

	CASE enStartUpStatus OF
		STRUP_DISABLED:
			IF gMachine.Pt.xAllowAutoStartUp AND gMachine.parSw.xAutoStartEnabled THEN
				enStartUpStatus := STRUP_NOT_STARTED;
			END_IF

		STRUP_NOT_STARTED:
			gMachine.St.StartUp.xReadyToAuto := FALSE;
			IF gMachine.St.Mode.xStartUp THEN
				//Sending a reset command to remove motor's error.
				//So when pressing reset to launch start up process (enPrinterState = PRINTERGEN_STARTUP when "EDGENEG(tofToAutoAfterEnableSafety.Q)")
				//safety relays are activated and STO restored to motor but a second reset is required in order to get those motor status ready to go
				IF gBlock[1].Status.Icla.xInError OR gBlock[1].Al.xAnyVerticalDriveAlarm THEN
					//To review how to send a reset order instead of using commandsSw reset
					gMachine.commandsSw.xReset_GI := TRUE;
				END_IF
				enStartUpStatus := STRUP_RESETTING_MOTORS;
			END_IF

		STRUP_RESETTING_MOTORS:
			gMachine.commandsSw.xReset_GI := FALSE;
			enStartUpStatus := STRUP_HOME_ICLA_ORDER;

		STRUP_HOME_ICLA_ORDER:
			gBlock[1].commands.xIclaHomeOrder := TRUE;
			IF gBlock[1].Status.Icla.xHoming THEN
				enStartUpStatus := STRUP_HOMING_ICLA;
			END_IF

		STRUP_HOMING_ICLA:
			IF gBlock[1].Status.Icla.xHomed THEN
				gBlock[1].commands.Manual.xManTrayOut := TRUE;
				enStartUpStatus := STRUP_MOVING_TRAY_OUT;
			END_IF

			IF gBlock[1].Status.Icla.xInError THEN
				enStartUpStatus := STRUP_ERROR;
			END_IF

		STRUP_MOVING_TRAY_OUT:
			IF gBlock[1].In.xTrayOut THEN
				gBlock[1].commands.xBarHomeOrder := TRUE;
				enStartUpStatus := STRUP_HOMING_BLOCK;
			END_IF

		STRUP_HOMING_BLOCK:
			//Once the block has been homed, with STARTUP the block is considered in AUTO
			IF gBlock[1].Status.Motor.xBarsHomed AND gBlock[1].Status.BlockState = BLOCK_AUTO THEN
				gBlock[1].commands.xToCap := TRUE;
				enStartUpStatus := STRUP_BLOCK_GOING_TO_CAP;
			END_IF

			IF gBlock[1].Al.xAlrReferenceIncoherence OR gBlock[1].Al.xAnyVerticalDriveAlarm THEN
				enStartUpStatus := STRUP_ERROR;
			END_IF

		STRUP_BLOCK_GOING_TO_CAP:
			IF gBlock[1].Status.Position.xInCap THEN
				gBlock[1].commands.Manual.xManTrayIn := TRUE;
				enStartUpStatus := STRUP_STARTING_INKS;
			END_IF

		STRUP_STARTING_INKS:
			// Start inks
			FOR iIndexStartUp := 1 TO gBlock[1].parameters.Inks.iMaxMachinePrintBars DO
				IF gInks[iIndexStartUp].parSw.Config.iMappingBar > 0 THEN
//					gInks[iIndexStartUp].parSw.Temp.rSetPointTemp := gInks[iIndexStartUp].parameters.parBar.Default.rTemp ;
//					gInks[iIndexStartUp].parSw.NegPump.rSetPointMeniscus := gInks[iIndexStartUp].parameters.parBar.StartUp.rMeniscus ;
//					gInks[iIndexStartUp].parSw.PosPump.rSetPoint := gInks[iIndexStartUp].parameters.parBar.StartUp.rPositive ;

					gInks[iIndexStartUp].parameters.StartUp.xActive := TRUE;
					gInks[iIndexStartUp].ordersSw.xStartInks := TRUE;
				END_IF
			END_FOR
			enStartUpStatus := STRUP_WAIT_INKS_STARTED;

		STRUP_WAIT_INKS_STARTED:
			tonStartingInks.IN := TRUE;
			tonStartingInks.PT := t#3s;
			tonStartingInks();
			IF tonStartingInks.Q THEN
				tonStartingInks(IN := FALSE); //Resetting timer
				enStartUpStatus := STRUP_REVIEWING_INKS;
			END_IF

		STRUP_REVIEWING_INKS:
			xStartUpAnyBarNotStable := FALSE; iIndexStartUp := 0;
			xStartUpAnyBarUnstable := FALSE;
			xInksStoppedWhileStartUp := FALSE;
			FOR iIndexStartUp := 1 TO gBlock[1].parameters.Inks.iMaxMachinePrintBars DO
				ReviewStartUpStatusInkIndex;
			END_FOR

			// If everyone is stable, go next step
			IF NOT xStartUpAnyBarNotStable THEN
				enStartUpStatus := STRUP_POWER_UP_PRINTHEADS;
			END_IF

			// If some bar is really unstable, cancel the startup
			IF xStartUpAnyBarUnstable AND xInksStoppedWhileStartUp THEN
				enStartUpStatus := STRUP_ERROR;
			END_IF

		STRUP_POWER_UP_PRINTHEADS:
			// Tutn on electronics
			FOR iIndexStartUp := 1 TO gBlock[1].parameters.Inks.iMaxMachinePrintBars DO
				IF gInks[iIndexStartUp].parSw.Config.iMappingBar > 0 THEN
					gInks[iIndexStartUp].ordersSw.xPowPrintHead := TRUE;
				END_IF
			END_FOR
			enStartUpStatus := STRUP_REVIEWING_PRINTHEADS;

		STRUP_REVIEWING_PRINTHEADS:
			xStartUpAnyBarNotPowered := FALSE;
			FOR iIndexStartUp := 1 TO gBlock[1].parameters.Inks.iMaxMachinePrintBars DO
				// Reviewing if the cards are turned on
				IF gInks[iIndexStartUp].parSw.Config.iMappingBar > 0 THEN
					IF NOT gInks[iIndexStartUp].signals.out.xOutPowPrintHead THEN
						xStartUpAnyBarNotPowered := TRUE;
					END_IF
				END_IF
			END_FOR

			IF NOT xStartUpAnyBarNotPowered THEN
				enStartUpStatus := STRUP_READY;
			END_IF

		STRUP_ERROR,
		STRUP_READY,
		STRUP_CANCELLED:
			gMachine.St.StartUp.xReadyToAuto := TRUE;

			// Assure in case of error or cancelled, the startup process in the inks is stopped
			FOR iIndexStartUp := 1 TO gBlock[1].parameters.Inks.iMaxMachinePrintBars DO
				gInks[iIndexStartUp].parameters.StartUp.xActive := FALSE;
			END_FOR

	END_CASE

	// Those are the states where cancel is blocked because make no sense
	xPosibleCancel.0 := enStartUpStatus = STRUP_ERROR;
	xPosibleCancel.1 := enStartUpStatus = STRUP_READY;
	xPosibleCancel.2 := enStartUpStatus = STRUP_CANCELLED;
	xPosibleCancel.3 := enStartUpStatus = STRUP_DISABLED;

	IF gMachine.commandsSw.xCancelStartUp AND xPosibleCancel = 0 THEN
		// Canceling homing icla if cancelled while homing
		IF enStartUpStatus = STRUP_HOMING_ICLA THEN
			gBlock[1].commands.xIclaHomeOrderInterrupt := TRUE;
		END_IF
		// Canceling homing bar if cancelled while homing
		IF enStartUpStatus = STRUP_HOMING_BLOCK THEN
			gBlock[1].commands.xBarHomeOrder := FALSE;
		END_IF
		enStartUpStatus := STRUP_CANCELLED;
	END_IF

	gMachine.St.StartUp.Status := enStartUpStatus;
	gMachine.St.StartUp.xInProgress := 	enStartUpStatus <> STRUP_DISABLED AND
										enStartUpStatus <> STRUP_NOT_STARTED AND
										enStartUpStatus <> STRUP_ERROR AND
										enStartUpStatus <> STRUP_READY AND
										enStartUpStatus <> STRUP_CANCELLED AND
										enStartUpStatus <> STRUP_DISABLED;

END_ACTION

ACTION ReviewStartUpStatusInkIndex:

	// If the bar cannot be started, do not consider it
	IF gInks[iIndexStartUp].parSw.Config.iMappingBar <= 0 THEN
		RETURN;
	END_IF

	// Running each inks system timer

	IF gInks[iIndexStartUp].status.AutoStartUp.xCancelled THEN
		// If detected a long unstability, change the set point to avoid stopping or dripping and raise the signal to go to error
		xStartUpAnyBarUnstable := TRUE;
	END_IF

	// Reviewing if the system is stable
	IF NOT gInks[iIndexStartUp].status.AutoStartUp.xStarted OR gInks[iIndexStartUp].Al.xAlrDiffInCtrlTemp OR gInks[iIndexStartUp].Al.xAlrDiffVacuum THEN
		xStartUpAnyBarNotStable := TRUE;
		iIndexBarNotStable := iIndexStartUp;
		UnstabInkStartUp[iIndexStartUp] := TRUE;
	ELSE
		UnstabInkStartUp[iIndexStartUp] := FALSE;
	END_IF

	IF NOT gInks[iIndexStartUp].status.xInksRunning THEN
		xInksStoppedWhileStartUp := TRUE;
	END_IF

END_ACTION
```

- StartUpProcessStates.graphml (not shown)

#### SuctionBlower.st
```iecst
ACTION SuctionBlower:

	////////////////////////////
	// BLOWERS
	////////////////////////////
	// Reference Jira: CRETAPRINT LEGOCRETALEGO-845
	// Turbine: Suction mode in automatic it isn´t correct.
	//
	// gui_i_iModoTurbina
	// Suction mode functionality. It can be configured by GUI with Ventrui or Turbine parameters
	// 0 estado off, 1 estado siempre On, modo 2, con base de tiempo en la desconexion.

	CASE gMachine.parSw.Suction.iBlowerMode OF

		BWMODE_OFF:
			xSuctionTurbine := FALSE;

		BWMODE_ON:
			xSuctionTurbine := TRUE;

		BWMODE_AUTO:
			IF NOT gMachine.Pt.xControlledByLine THEN
				tofDelaySuction.IN:=gMachine.St.Mode.xAuto AND gBelt.states.xRuningBelt;
				tofDelaySuction.PT:=gMachine.parSw.Suction.tiBlowerDelayOff;
				tofDelaySuction();

				xSuctionTurbine := tofDelaySuction.Q;

			ELSE
				//[RGP] To be discussed with controls team. I think this is a better solution for mist collector
				tofDelaySuction.IN:= (NOT gBelt.states.xRuningBelt) OR (NOT gThicknessCtrl.status.MediaPosition.xMediaInside) ;
				tofDelaySuction.PT:=gMachine.parSw.Suction.tiBlowerDelayOff;
				tofDelaySuction();

				rsSuction.RESET1 := tofDelaySuction.Q;
				rsSuction.SET := gThicknessCtrl.status.MediaPosition.xMediaInside;
				rsSuction();

				xSuctionTurbine := rsSuction.Q1;
			END_IF
	END_CASE

	gMachine.Out.xSuctionTurbine := xSuctionTurbine AND NOT gMachine.In.xHoppersSoftStarterFault;

END_ACTION
```

### Program Logical/Printer/MachineCtrl/MachineCtrl_Fast (IEC) - Machine program

#### Alarms.st
```iecst
ACTION Alarms:

	// Warning Alarm raised when a new BentTile is detected. The signal is kept for 5s
	TP_AlrBentTile.IN:=(gMachine.St.AutoMode.xProdORLab AND EDGEPOS(gThicknessCtrl.status.Heigh.xIncreasedHeigh[1]) AND (NOT xMediaThicknessModified));
	TP_AlrBentTile.PT:= T#5S;
	TP_AlrBentTile();
	gMachine.Al.Warning.xBentTile:=TP_AlrBentTile.Q;

	// Copy new thickness value
	IF TP_AlrBentTile.Q OR EDGENEG(gThicknessCtrl.status.Heigh.xIncreasedHeigh[1]) OR EDGEPOS(gMachine.St.AutoMode.xProdORLab)THEN
		rPrevMediaThickness := gMachine.parSw.Media.rThickness;
	END_IF

	// Alarm: No bars in Print
	IF	(NOT gMachine.St.Position.xInPrint AND gMachine.St.AutoMode.xProduction AND
		EDGEPOS(gThicknessCtrl.Outputs.xMediaFiltered) AND (NOT gLine.StatusSummary.xEmptyingBelts)) THEN
		gMachine.Al.Alarm.xAlarmNotInPrintPosition:=TRUE;
	ELSIF gMachine.St.Mode.xZero OR (gMachine.St.Position.xInPrint AND gMachine.St.AutoMode.xProdORLab) THEN // Is it gMachine.St.Position.xInPrint or zero state?
		gMachine.Al.Alarm.xAlarmNotInPrintPosition:=FALSE;
	END_IF

	//Low bat + Power Fault = Power Off
	IF gMachine.Al.Alarm.xAlarmSAIPowerFault AND (gMachine.In.UPSs[1].xLowBattery OR (gMachine.In.UPSs[2].xLowBattery AND (gMachine.Pt.CT.iNumBlocks>=2))) THEN
		gMachine.Al.Alarm.xAlarmSAIPowerOff:= TRUE;
	END_IF

	//24VDC Power Supply for IDS
	IF NOT gMachine.In.x24Vdc THEN gMachine.Al.Alarm.xAlr24Vdc := TRUE; END_IF

	//Alarm: Mounted Piece Inide the Machine
	IF (gPhotoCells.Alarms.xMountedTile OR gDing.Alarms.xMountedTile OR gBasicDetectMedia.Alarms.xMountedMedia) THEN
		gMachine.Al.Alarm.xAlarmMountedPiece:= TRUE;
	END_IF

	gMachine.Al.Warning.xMountedMediaInside := gThicknessCtrl.status.MediaPosition.xMountedMediaInside;

	//Degasser
	TON_AlrDegasserPressure(IN:=gMachine.Out.xDegasser AND NOT gMachine.In.xDegasserPressure, PT:=T#3S);
	IF TON_AlrDegasserPressure.Q THEN gMachine.Al.Warning.xAlrDegasserPressure:=TRUE; END_IF

	//Alarm: Broken PD
	IF NOT gThicknessCtrl.parameters.Detection.Array.xLoadMedia THEN CalcPDSensorAlarm; END_IF

	//Ding wrong position
	WrongDingPosition;

	//Alarm: Sw reports a critical condition to execute printing process
    IF gMachine.parSw.UI.xCriticalCondition THEN
        IF gMachine.Pt.xControlledByLine AND gLine.StatusSummary.xPrinting THEN
            gMachine.Al.Alarm.xSwCriticalCondition := TRUE;
        END_IF
    END_IF

	//Incoherence between sensors array and product detect. DELOREAN-2709
	IF gMachine.St.Position.xInPrint THEN
		IF EDGEPOS(gThicknessCtrl.status.MediaPosition.L1.xDetectionSystemIncoherence) THEN
			gMachine.Al.Warning.xMediaIncoherenceDetectedL1:=TRUE;
		END_IF

		IF gMachine.parSw.Dtp.xDoubleLine AND EDGEPOS(gThicknessCtrl.status.MediaPosition.L2.xDetectionSystemIncoherence) THEN
			gMachine.Al.Warning.xMediaIncoherenceDetectedL2:=TRUE;
		END_IF
	END_IF

	gMachine.Al.Alarm.xAlrSafetyNotEnabled := NOT gMachine.In.xSafetyEnabled;

END_ACTION

ACTION CalcPDSensorAlarm:

	//When no sensor is connected, cannot be checked
	IF (gMachine.Pt.PDSignalTpe <> PDCFG_SENSOR AND gMachine.Pt.PDSignalTpe <> PDCFG_SENSOR_AND_CARRIAGE) THEN
		gMachine.Lg.udiPiecesCounterErrorL1 := 0;
		gMachine.Lg.udiPiecesCounterErrorL2 := 0;
		RETURN;
	END_IF

	//Reset counter when belt is stoped or not in printin
	IF NOT gBelt.states.xRuningBelt OR NOT gMachine.St.Position.xInPrint THEN
		gMachine.Lg.udiPiecesCounterErrorL1 := 0;
		gMachine.Lg.udiPiecesCounterErrorL2 := 0;
		RETURN;
	END_IF

	//Sensor 1
	xEnabledAlarmPDSensor1 := NOT gMachine.parSw.Dtp.xDoubleLine OR (gMachine.parSw.Dtp.xDoubleLine AND gMachine.parSw.Dtp.iModeLine1 = GC_DTP_RUN AND gMachine.parSw.Dtp.iModeLine2 = GC_DTP_STOP);
	T_AlarmPDL1.IN:= NOT gMachine.Pt.ProductDetect.xDisableBrokenSensor AND xEnabledAlarmPDSensor1 AND NOT gMachine.St.ProductDetect.xProductDetectL1 AND gMachine.St.xMediaDetected;						//If Photocell1 Detect Tile and PD not
	IF gBelt.states.rCurrentSpeed > 0 THEN
		T_AlarmPDL1.PT:= REAL_TO_TIME( 60 * (gMachine.Pt.CT.rDistanceThicknesToPD + 8) / gBelt.states.rCurrentSpeed);		//In a time (depends of belt speed and distance between sensors). Adding 8mm safety
	END_IF
	T_AlarmPDL1();
	IF EDGEPOS(T_AlarmPDL1.Q) THEN gMachine.Lg.udiPiecesCounterErrorL1 := gMachine.Lg.udiPiecesCounterErrorL1 + 1; END_IF	//Increase Error Detect Counter

	IF gMachine.Pt.Hw.xDoubleLineAllowed THEN
		//Sensor 2
		xEnabledAlarmPDSensor2 := gMachine.parSw.Dtp.xDoubleLine AND gMachine.parSw.Dtp.iModeLine1 = GC_DTP_STOP AND gMachine.parSw.Dtp.iModeLine2 = GC_DTP_RUN;
		T_AlarmPDL2.IN:= NOT gMachine.Pt.ProductDetect.xDisableBrokenSensor AND xEnabledAlarmPDSensor2 AND NOT xPDSignalSensorL2 AND gMachine.St.xMediaDetected;
		IF gBelt.states.rCurrentSpeed > 0 THEN
			T_AlarmPDL2.PT:= REAL_TO_TIME( 60 * (gMachine.Pt.CT.rDistanceThicknesToPD + 8) / gBelt.states.rCurrentSpeed);		//In a time (depends of belt speed and distance between sensors). Adding 8mm safety
		END_IF
		T_AlarmPDL2();
		IF EDGEPOS(T_AlarmPDL2.Q) THEN gMachine.Lg.udiPiecesCounterErrorL2 := gMachine.Lg.udiPiecesCounterErrorL2 + 1; END_IF
	END_IF

//	IF gMachine.Lg.udiPiecesCounterErrorL1 > 10 THEN gMachine.Al.Alarm.xPDBrokenSensorL1:= TRUE; END_IF
//	IF gMachine.Lg.udiPiecesCounterErrorL2 > 10 THEN gMachine.Al.Alarm.xPDBrokenSensorL2:= TRUE; END_IF

END_ACTION

ACTION WrongDingPosition:

	IF NOT gDing.State.xDingInstalled OR NOT gDing.Parameters.xRaiseDigitalIncoherency THEN
		RETURN;
	END_IF

	//Protect the code of a Zero division
	IF gBelt.states.rCurrentSpeed < 0.1 THEN
		TOF_AlarmDingPosition.IN := FALSE;
		TOF_AlarmDingPosition();
		RETURN;
	END_IF

	TOF_AlarmDingPosition.IN := gDing.State.xDingLowPieceDetect;
	IF gBelt.states.rCurrentSpeed > 0 THEN
		TOF_AlarmDingPosition.PT := REAL_TO_TIME( 60 * (gMachine.Pt.CT.rDistanceThicknesToPD + 8) / gBelt.states.rCurrentSpeed);
	END_IF
	TOF_AlarmDingPosition();

	xPrintShootingForced := gMachine.Out.xShotLine1 OR gMachine.Out.xShotLine2;
	IF	NOT TOF_AlarmDingPosition.Q AND NOT xPrintShootingForced AND gBelt.states.xRuningBelt AND
		gMachine.St.AutoMode.xProdORLab AND EDGEPOS(gMachine.St.ProductDetect.xAnyProductDetectDtpStricted) THEN

		gMachine.Al.Alarm.xAlrDingWrongPosition := TRUE;
	END_IF

END_ACTION
```
